# B&R Automation Studio project CleanChemi_SiteManagementSystem (part 7)

```iecst
		IF gSkid_LR[IdxSkids_LR].Alarms.ALARM_AB15.4 AND gServices.Alarms_LR[IdxSkids_LR].Internal.Alarms_State.ALARM_AB15.4 = FALSE THEN
			IF gSkid_LR[IdxSkids_LR].ErrorInfo.Text = '' THEN
				gSkid_LR[IdxSkids_LR].ErrorInfo.Text		:= 'ALARM_AB15.4';
				gSkid_LR[IdxSkids_LR].ErrorInfo.State		:= 'Warning';
				gSkid_LR[IdxSkids_LR].ErrorInfo.Severity	:= 1;
				gSkid_LR[IdxSkids_LR].Error := TRUE;
				gServices.Alarms_LR[IdxSkids_LR].Internal.Alarms_State.ALARM_AB15.4 := TRUE;
			END_IF
		END_IF;

		IF gSkid_LR[IdxSkids_LR].Alarms.ALARM_AB15.5 AND gServices.Alarms_LR[IdxSkids_LR].Internal.Alarms_State.ALARM_AB15.5 = FALSE THEN
			IF gSkid_LR[IdxSkids_LR].ErrorInfo.Text = '' THEN
				gSkid_LR[IdxSkids_LR].ErrorInfo.Text		:= 'ALARM_AB15.5';
				gSkid_LR[IdxSkids_LR].ErrorInfo.State		:= 'Warning';
				gSkid_LR[IdxSkids_LR].ErrorInfo.Severity	:= 1;
				gSkid_LR[IdxSkids_LR].Error := TRUE;
				gServices.Alarms_LR[IdxSkids_LR].Internal.Alarms_State.ALARM_AB15.5 := TRUE;
			END_IF
		END_IF;

		IF gSkid_LR[IdxSkids_LR].Alarms.ALARM_AB15.6 AND gServices.Alarms_LR[IdxSkids_LR].Internal.Alarms_State.ALARM_AB15.6 = FALSE THEN
			IF gSkid_LR[IdxSkids_LR].ErrorInfo.Text = '' THEN
				gSkid_LR[IdxSkids_LR].ErrorInfo.Text		:= 'ALARM_AB15.6';
				gSkid_LR[IdxSkids_LR].ErrorInfo.State		:= 'Warning';
				gSkid_LR[IdxSkids_LR].ErrorInfo.Severity	:= 1;
				gSkid_LR[IdxSkids_LR].Error := TRUE;
				gServices.Alarms_LR[IdxSkids_LR].Internal.Alarms_State.ALARM_AB15.6 := TRUE;
			END_IF
		END_IF;
		IF gSkid_LR[IdxSkids_LR].Alarms.ALARM_AB15.7 AND gServices.Alarms_LR[IdxSkids_LR].Internal.Alarms_State.ALARM_AB15.7 = FALSE THEN
			IF gSkid_LR[IdxSkids_LR].ErrorInfo.Text = '' THEN
				gSkid_LR[IdxSkids_LR].ErrorInfo.Text		:= 'ALARM_AB15.7';
				gSkid_LR[IdxSkids_LR].ErrorInfo.State		:= 'Warning';
				gSkid_LR[IdxSkids_LR].ErrorInfo.Severity	:= 1;
				gSkid_LR[IdxSkids_LR].Error := TRUE;
				gServices.Alarms_LR[IdxSkids_LR].Internal.Alarms_State.ALARM_AB15.7 := TRUE;
			END_IF
		END_IF;
		IF gSkid_LR[IdxSkids_LR].Alarms.ALARM_AB15.8 AND gServices.Alarms_LR[IdxSkids_LR].Internal.Alarms_State.ALARM_AB15.8 = FALSE THEN
			IF gSkid_LR[IdxSkids_LR].ErrorInfo.Text = '' THEN
				gSkid_LR[IdxSkids_LR].ErrorInfo.Text		:= 'ALARM_AB15.8';
				gSkid_LR[IdxSkids_LR].ErrorInfo.State		:= 'Warning';
				gSkid_LR[IdxSkids_LR].ErrorInfo.Severity	:= 1;
				gSkid_LR[IdxSkids_LR].Error := TRUE;
				gServices.Alarms_LR[IdxSkids_LR].Internal.Alarms_State.ALARM_AB15.8 := TRUE;
			END_IF
		END_IF;
		IF gSkid_LR[IdxSkids_LR].Alarms.ALARM_AB15.9 AND gServices.Alarms_LR[IdxSkids_LR].Internal.Alarms_State.ALARM_AB15.9 = FALSE THEN
			IF gSkid_LR[IdxSkids_LR].ErrorInfo.Text = '' THEN
				gSkid_LR[IdxSkids_LR].ErrorInfo.Text		:= 'ALARM_AB15.9';
				gSkid_LR[IdxSkids_LR].ErrorInfo.State		:= 'Warning';
				gSkid_LR[IdxSkids_LR].ErrorInfo.Severity	:= 1;
				gSkid_LR[IdxSkids_LR].Error := TRUE;
				gServices.Alarms_LR[IdxSkids_LR].Internal.Alarms_State.ALARM_AB15.9 := TRUE;
			END_IF
		END_IF;
		IF gSkid_LR[IdxSkids_LR].Alarms.ALARM_AB15.10 AND gServices.Alarms_LR[IdxSkids_LR].Internal.Alarms_State.ALARM_AB15.10 = FALSE THEN
			IF gSkid_LR[IdxSkids_LR].ErrorInfo.Text = '' THEN
				gSkid_LR[IdxSkids_LR].ErrorInfo.Text		:= 'ALARM_AB15.10';
				gSkid_LR[IdxSkids_LR].ErrorInfo.State		:= 'Warning';
				gSkid_LR[IdxSkids_LR].ErrorInfo.Severity	:= 1;
				gSkid_LR[IdxSkids_LR].Error := TRUE;
				gServices.Alarms_LR[IdxSkids_LR].Internal.Alarms_State.ALARM_AB15.10 := TRUE;
			END_IF
		END_IF;
		IF gSkid_LR[IdxSkids_LR].Alarms.ALARM_AB15.11 AND gServices.Alarms_LR[IdxSkids_LR].Internal.Alarms_State.ALARM_AB15.11 = FALSE THEN
			IF gSkid_LR[IdxSkids_LR].ErrorInfo.Text = '' THEN
				gSkid_LR[IdxSkids_LR].ErrorInfo.Text		:= 'ALARM_AB15.11';
				gSkid_LR[IdxSkids_LR].ErrorInfo.State		:= 'Warning';
				gSkid_LR[IdxSkids_LR].ErrorInfo.Severity	:= 1;
				gSkid_LR[IdxSkids_LR].Error := TRUE;
				gServices.Alarms_LR[IdxSkids_LR].Internal.Alarms_State.ALARM_AB15.11 := TRUE;
			END_IF
		END_IF;
		IF gSkid_LR[IdxSkids_LR].Alarms.ALARM_AB15.12 AND gServices.Alarms_LR[IdxSkids_LR].Internal.Alarms_State.ALARM_AB15.12 = FALSE THEN
			IF gSkid_LR[IdxSkids_LR].ErrorInfo.Text = '' THEN
				gSkid_LR[IdxSkids_LR].ErrorInfo.Text		:= 'ALARM_AB15.12';
				gSkid_LR[IdxSkids_LR].ErrorInfo.State		:= 'Warning';
				gSkid_LR[IdxSkids_LR].ErrorInfo.Severity	:= 1;
				gSkid_LR[IdxSkids_LR].Error := TRUE;
				gServices.Alarms_LR[IdxSkids_LR].Internal.Alarms_State.ALARM_AB15.12 := TRUE;
			END_IF
		END_IF;

		// AB16
		IF gSkid_LR[IdxSkids_LR].Alarms.ALARM_AB16.0 AND gServices.Alarms_LR[IdxSkids_LR].Internal.Alarms_State.ALARM_AB16.0 = FALSE THEN
			IF gSkid_LR[IdxSkids_LR].ErrorInfo.Text = '' THEN
				gSkid_LR[IdxSkids_LR].ErrorInfo.Text		:= 'ALARM_AB16.0';
				gSkid_LR[IdxSkids_LR].ErrorInfo.State		:= 'Warning';
				gSkid_LR[IdxSkids_LR].ErrorInfo.Severity	:= 2;
				gSkid_LR[IdxSkids_LR].Error := TRUE;
				gServices.Alarms_LR[IdxSkids_LR].Internal.Alarms_State.ALARM_AB16.0 := TRUE;
			END_IF
		END_IF;

		IF gSkid_LR[IdxSkids_LR].Alarms.ALARM_AB16.1 AND gServices.Alarms_LR[IdxSkids_LR].Internal.Alarms_State.ALARM_AB16.1 = FALSE THEN
			IF gSkid_LR[IdxSkids_LR].ErrorInfo.Text = '' THEN
				gSkid_LR[IdxSkids_LR].ErrorInfo.Text		:= 'ALARM_AB16.1';
				gSkid_LR[IdxSkids_LR].ErrorInfo.State		:= 'Warning';
				gSkid_LR[IdxSkids_LR].ErrorInfo.Severity	:= 1;
				gSkid_LR[IdxSkids_LR].Error := TRUE;
				gServices.Alarms_LR[IdxSkids_LR].Internal.Alarms_State.ALARM_AB16.1 := TRUE;
			END_IF
		END_IF;

		IF gSkid_LR[IdxSkids_LR].Alarms.ALARM_AB16.2 AND gServices.Alarms_LR[IdxSkids_LR].Internal.Alarms_State.ALARM_AB16.2 = FALSE THEN
			IF gSkid_LR[IdxSkids_LR].ErrorInfo.Text = '' THEN
				gSkid_LR[IdxSkids_LR].ErrorInfo.Text		:= 'ALARM_AB16.2';
				gSkid_LR[IdxSkids_LR].ErrorInfo.State		:= 'Warning';
				gSkid_LR[IdxSkids_LR].ErrorInfo.Severity	:= 2;
				gSkid_LR[IdxSkids_LR].Error := TRUE;
				gServices.Alarms_LR[IdxSkids_LR].Internal.Alarms_State.ALARM_AB16.2 := TRUE;
			END_IF
		END_IF;

		IF gSkid_LR[IdxSkids_LR].Alarms.ALARM_AB16.3 AND gServices.Alarms_LR[IdxSkids_LR].Internal.Alarms_State.ALARM_AB16.3 = FALSE THEN
			IF gSkid_LR[IdxSkids_LR].ErrorInfo.Text = '' THEN
				gSkid_LR[IdxSkids_LR].ErrorInfo.Text		:= 'ALARM_AB16.3';
				gSkid_LR[IdxSkids_LR].ErrorInfo.State		:= 'Warning';
				gSkid_LR[IdxSkids_LR].ErrorInfo.Severity	:= 1;
				gSkid_LR[IdxSkids_LR].Error := TRUE;
				gServices.Alarms_LR[IdxSkids_LR].Internal.Alarms_State.ALARM_AB16.3 := TRUE;
			END_IF
		END_IF;

		IF gSkid_LR[IdxSkids_LR].Alarms.ALARM_AB16.4 AND gServices.Alarms_LR[IdxSkids_LR].Internal.Alarms_State.ALARM_AB16.4 = FALSE THEN
			IF gSkid_LR[IdxSkids_LR].ErrorInfo.Text = '' THEN
				gSkid_LR[IdxSkids_LR].ErrorInfo.Text		:= 'ALARM_AB16.4';
				gSkid_LR[IdxSkids_LR].ErrorInfo.State		:= 'Warning';
				gSkid_LR[IdxSkids_LR].ErrorInfo.Severity	:= 2;
				gSkid_LR[IdxSkids_LR].Error := TRUE;
				gServices.Alarms_LR[IdxSkids_LR].Internal.Alarms_State.ALARM_AB16.4 := TRUE;
			END_IF
		END_IF;

		IF gSkid_LR[IdxSkids_LR].Alarms.ALARM_AB16.5 AND gServices.Alarms_LR[IdxSkids_LR].Internal.Alarms_State.ALARM_AB16.5 = FALSE THEN
			IF gSkid_LR[IdxSkids_LR].ErrorInfo.Text = '' THEN
				gSkid_LR[IdxSkids_LR].ErrorInfo.Text		:= 'ALARM_AB16.5';
				gSkid_LR[IdxSkids_LR].ErrorInfo.State		:= 'Warning';
				gSkid_LR[IdxSkids_LR].ErrorInfo.Severity	:= 1;
				gSkid_LR[IdxSkids_LR].Error := TRUE;
				gServices.Alarms_LR[IdxSkids_LR].Internal.Alarms_State.ALARM_AB16.5 := TRUE;
			END_IF
		END_IF;

		IF gSkid_LR[IdxSkids_LR].Alarms.ALARM_AB16.6 AND gServices.Alarms_LR[IdxSkids_LR].Internal.Alarms_State.ALARM_AB16.6 = FALSE THEN
			IF gSkid_LR[IdxSkids_LR].ErrorInfo.Text = '' THEN
				gSkid_LR[IdxSkids_LR].ErrorInfo.Text		:= 'ALARM_AB16.6';
				gSkid_LR[IdxSkids_LR].ErrorInfo.State		:= 'Warning';
				gSkid_LR[IdxSkids_LR].ErrorInfo.Severity	:= 2;
				gSkid_LR[IdxSkids_LR].Error := TRUE;
				gServices.Alarms_LR[IdxSkids_LR].Internal.Alarms_State.ALARM_AB16.6 := TRUE;
			END_IF
		END_IF;
		IF gSkid_LR[IdxSkids_LR].Alarms.ALARM_AB16.7 AND gServices.Alarms_LR[IdxSkids_LR].Internal.Alarms_State.ALARM_AB16.7 = FALSE THEN
			IF gSkid_LR[IdxSkids_LR].ErrorInfo.Text = '' THEN
				gSkid_LR[IdxSkids_LR].ErrorInfo.Text		:= 'ALARM_AB16.7';
				gSkid_LR[IdxSkids_LR].ErrorInfo.State		:= 'Warning';
				gSkid_LR[IdxSkids_LR].ErrorInfo.Severity	:= 1;
				gSkid_LR[IdxSkids_LR].Error := TRUE;
				gServices.Alarms_LR[IdxSkids_LR].Internal.Alarms_State.ALARM_AB16.7 := TRUE;
			END_IF
		END_IF;
		IF gSkid_LR[IdxSkids_LR].Alarms.ALARM_AB16.8 AND gServices.Alarms_LR[IdxSkids_LR].Internal.Alarms_State.ALARM_AB16.8 = FALSE THEN
			IF gSkid_LR[IdxSkids_LR].ErrorInfo.Text = '' THEN
				gSkid_LR[IdxSkids_LR].ErrorInfo.Text		:= 'ALARM_AB16.8';
				gSkid_LR[IdxSkids_LR].ErrorInfo.State		:= 'Warning';
				gSkid_LR[IdxSkids_LR].ErrorInfo.Severity	:= 2;
				gSkid_LR[IdxSkids_LR].Error := TRUE;
				gServices.Alarms_LR[IdxSkids_LR].Internal.Alarms_State.ALARM_AB16.8 := TRUE;
			END_IF
		END_IF;
		IF gSkid_LR[IdxSkids_LR].Alarms.ALARM_AB16.9 AND gServices.Alarms_LR[IdxSkids_LR].Internal.Alarms_State.ALARM_AB16.9 = FALSE THEN
			IF gSkid_LR[IdxSkids_LR].ErrorInfo.Text = '' THEN
				gSkid_LR[IdxSkids_LR].ErrorInfo.Text		:= 'ALARM_AB16.9';
				gSkid_LR[IdxSkids_LR].ErrorInfo.State		:= 'Warning';
				gSkid_LR[IdxSkids_LR].ErrorInfo.Severity	:= 1;
				gSkid_LR[IdxSkids_LR].Error := TRUE;
				gServices.Alarms_LR[IdxSkids_LR].Internal.Alarms_State.ALARM_AB16.9 := TRUE;
			END_IF
		END_IF;
		IF gSkid_LR[IdxSkids_LR].Alarms.ALARM_AB16.10 AND gServices.Alarms_LR[IdxSkids_LR].Internal.Alarms_State.ALARM_AB16.10 = FALSE THEN
			IF gSkid_LR[IdxSkids_LR].ErrorInfo.Text = '' THEN
				gSkid_LR[IdxSkids_LR].ErrorInfo.Text		:= 'ALARM_AB16.10';
				gSkid_LR[IdxSkids_LR].ErrorInfo.State		:= 'Warning';
				gSkid_LR[IdxSkids_LR].ErrorInfo.Severity	:= 2;
				gSkid_LR[IdxSkids_LR].Error := TRUE;
				gServices.Alarms_LR[IdxSkids_LR].Internal.Alarms_State.ALARM_AB16.10 := TRUE;
			END_IF
		END_IF;
		IF gSkid_LR[IdxSkids_LR].Alarms.ALARM_AB16.11 AND gServices.Alarms_LR[IdxSkids_LR].Internal.Alarms_State.ALARM_AB16.11 = FALSE THEN
			IF gSkid_LR[IdxSkids_LR].ErrorInfo.Text = '' THEN
				gSkid_LR[IdxSkids_LR].ErrorInfo.Text		:= 'ALARM_AB16.11';
				gSkid_LR[IdxSkids_LR].ErrorInfo.State		:= 'Warning';
				gSkid_LR[IdxSkids_LR].ErrorInfo.Severity	:= 1;
				gSkid_LR[IdxSkids_LR].Error := TRUE;
				gServices.Alarms_LR[IdxSkids_LR].Internal.Alarms_State.ALARM_AB16.11 := TRUE;
			END_IF
		END_IF;
		IF gSkid_LR[IdxSkids_LR].Alarms.ALARM_AB16.12 AND gServices.Alarms_LR[IdxSkids_LR].Internal.Alarms_State.ALARM_AB16.12 = FALSE THEN
			IF gSkid_LR[IdxSkids_LR].ErrorInfo.Text = '' THEN
				gSkid_LR[IdxSkids_LR].ErrorInfo.Text		:= 'ALARM_AB16.12';
				gSkid_LR[IdxSkids_LR].ErrorInfo.State		:= 'Warning';
				gSkid_LR[IdxSkids_LR].ErrorInfo.Severity	:= 2;
				gSkid_LR[IdxSkids_LR].Error := TRUE;
				gServices.Alarms_LR[IdxSkids_LR].Internal.Alarms_State.ALARM_AB16.12 := TRUE;
			END_IF
		END_IF;
		IF gSkid_LR[IdxSkids_LR].Alarms.ALARM_AB16.13 AND gServices.Alarms_LR[IdxSkids_LR].Internal.Alarms_State.ALARM_AB16.13 = FALSE THEN
			IF gSkid_LR[IdxSkids_LR].ErrorInfo.Text = '' THEN
				gSkid_LR[IdxSkids_LR].ErrorInfo.Text		:= 'ALARM_AB16.13';
				gSkid_LR[IdxSkids_LR].ErrorInfo.State		:= 'Warning';
				gSkid_LR[IdxSkids_LR].ErrorInfo.Severity	:= 1;
				gSkid_LR[IdxSkids_LR].Error := TRUE;
				gServices.Alarms_LR[IdxSkids_LR].Internal.Alarms_State.ALARM_AB16.13 := TRUE;
			END_IF
		END_IF;
		IF gSkid_LR[IdxSkids_LR].Alarms.ALARM_AB16.14 AND gServices.Alarms_LR[IdxSkids_LR].Internal.Alarms_State.ALARM_AB16.14 = FALSE THEN
			IF gSkid_LR[IdxSkids_LR].ErrorInfo.Text = '' THEN
				gSkid_LR[IdxSkids_LR].ErrorInfo.Text		:= 'ALARM_AB16.14';
				gSkid_LR[IdxSkids_LR].ErrorInfo.State		:= 'Warning';
				gSkid_LR[IdxSkids_LR].ErrorInfo.Severity	:= 2;
				gSkid_LR[IdxSkids_LR].Error := TRUE;
				gServices.Alarms_LR[IdxSkids_LR].Internal.Alarms_State.ALARM_AB16.14 := TRUE;
			END_IF
		END_IF;
		IF gSkid_LR[IdxSkids_LR].Alarms.ALARM_AB16.15 AND gServices.Alarms_LR[IdxSkids_LR].Internal.Alarms_State.ALARM_AB16.15 = FALSE THEN
			IF gSkid_LR[IdxSkids_LR].ErrorInfo.Text = '' THEN
				gSkid_LR[IdxSkids_LR].ErrorInfo.Text		:= 'ALARM_AB16.15';
				gSkid_LR[IdxSkids_LR].ErrorInfo.State		:= 'Warning';
				gSkid_LR[IdxSkids_LR].ErrorInfo.Severity	:= 1;
				gSkid_LR[IdxSkids_LR].Error := TRUE;
				gServices.Alarms_LR[IdxSkids_LR].Internal.Alarms_State.ALARM_AB16.15 := TRUE;
			END_IF
		END_IF;

		// AB17
		IF gSkid_LR[IdxSkids_LR].Alarms.ALARM_AB17.0 AND gServices.Alarms_LR[IdxSkids_LR].Internal.Alarms_State.ALARM_AB17.0 = FALSE THEN
			IF gSkid_LR[IdxSkids_LR].ErrorInfo.Text = '' THEN
				gSkid_LR[IdxSkids_LR].ErrorInfo.Text		:= 'ALARM_AB17.0';
				gSkid_LR[IdxSkids_LR].ErrorInfo.State		:= 'Warning';
				gSkid_LR[IdxSkids_LR].ErrorInfo.Severity	:= 2;
				gSkid_LR[IdxSkids_LR].Error := TRUE;
				gServices.Alarms_LR[IdxSkids_LR].Internal.Alarms_State.ALARM_AB17.0 := TRUE;
			END_IF
		END_IF;

		IF gSkid_LR[IdxSkids_LR].Alarms.ALARM_AB17.1 AND gServices.Alarms_LR[IdxSkids_LR].Internal.Alarms_State.ALARM_AB17.1 = FALSE THEN
			IF gSkid_LR[IdxSkids_LR].ErrorInfo.Text = '' THEN
				gSkid_LR[IdxSkids_LR].ErrorInfo.Text		:= 'ALARM_AB17.1';
				gSkid_LR[IdxSkids_LR].ErrorInfo.State		:= 'Warning';
				gSkid_LR[IdxSkids_LR].ErrorInfo.Severity	:= 1;
				gSkid_LR[IdxSkids_LR].Error := TRUE;
				gServices.Alarms_LR[IdxSkids_LR].Internal.Alarms_State.ALARM_AB17.1 := TRUE;
			END_IF
		END_IF;

		IF gSkid_LR[IdxSkids_LR].Alarms.ALARM_AB17.2 AND gServices.Alarms_LR[IdxSkids_LR].Internal.Alarms_State.ALARM_AB17.2 = FALSE THEN
			IF gSkid_LR[IdxSkids_LR].ErrorInfo.Text = '' THEN
				gSkid_LR[IdxSkids_LR].ErrorInfo.Text		:= 'ALARM_AB17.2';
				gSkid_LR[IdxSkids_LR].ErrorInfo.State		:= 'Warning';
				gSkid_LR[IdxSkids_LR].ErrorInfo.Severity	:= 1;
				gSkid_LR[IdxSkids_LR].Error := TRUE;
				gServices.Alarms_LR[IdxSkids_LR].Internal.Alarms_State.ALARM_AB17.2 := TRUE;
			END_IF
		END_IF;

		IF gSkid_LR[IdxSkids_LR].Alarms.ALARM_AB17.3 AND gServices.Alarms_LR[IdxSkids_LR].Internal.Alarms_State.ALARM_AB17.3 = FALSE THEN
			IF gSkid_LR[IdxSkids_LR].ErrorInfo.Text = '' THEN
				gSkid_LR[IdxSkids_LR].ErrorInfo.Text		:= 'ALARM_AB17.3';
				gSkid_LR[IdxSkids_LR].ErrorInfo.State		:= 'Warning';
				gSkid_LR[IdxSkids_LR].ErrorInfo.Severity	:= 1;
				gSkid_LR[IdxSkids_LR].Error := TRUE;
				gServices.Alarms_LR[IdxSkids_LR].Internal.Alarms_State.ALARM_AB17.3 := TRUE;
			END_IF
		END_IF;

		IF gSkid_LR[IdxSkids_LR].Alarms.ALARM_AB17.4 AND gServices.Alarms_LR[IdxSkids_LR].Internal.Alarms_State.ALARM_AB17.4 = FALSE THEN
			IF gSkid_LR[IdxSkids_LR].ErrorInfo.Text = '' THEN
				gSkid_LR[IdxSkids_LR].ErrorInfo.Text		:= 'ALARM_AB17.4';
				gSkid_LR[IdxSkids_LR].ErrorInfo.State		:= 'Warning';
				gSkid_LR[IdxSkids_LR].ErrorInfo.Severity	:= 1;
				gSkid_LR[IdxSkids_LR].Error := TRUE;
				gServices.Alarms_LR[IdxSkids_LR].Internal.Alarms_State.ALARM_AB17.4 := TRUE;
			END_IF
		END_IF;

		IF gSkid_LR[IdxSkids_LR].Alarms.ALARM_AB17.5 AND gServices.Alarms_LR[IdxSkids_LR].Internal.Alarms_State.ALARM_AB17.5 = FALSE THEN
			IF gSkid_LR[IdxSkids_LR].ErrorInfo.Text = '' THEN
				gSkid_LR[IdxSkids_LR].ErrorInfo.Text		:= 'ALARM_AB17.5';
				gSkid_LR[IdxSkids_LR].ErrorInfo.State		:= 'Warning';
				gSkid_LR[IdxSkids_LR].ErrorInfo.Severity	:= 1;
				gSkid_LR[IdxSkids_LR].Error := TRUE;
				gServices.Alarms_LR[IdxSkids_LR].Internal.Alarms_State.ALARM_AB17.5 := TRUE;
			END_IF
		END_IF;

		IF gSkid_LR[IdxSkids_LR].Alarms.ALARM_AB17.6 AND gServices.Alarms_LR[IdxSkids_LR].Internal.Alarms_State.ALARM_AB17.6 = FALSE THEN
			IF gSkid_LR[IdxSkids_LR].ErrorInfo.Text = '' THEN
				gSkid_LR[IdxSkids_LR].ErrorInfo.Text		:= 'ALARM_AB17.6';
				gSkid_LR[IdxSkids_LR].ErrorInfo.State		:= 'Warning';
				gSkid_LR[IdxSkids_LR].ErrorInfo.Severity	:= 1;
				gSkid_LR[IdxSkids_LR].Error := TRUE;
				gServices.Alarms_LR[IdxSkids_LR].Internal.Alarms_State.ALARM_AB17.6 := TRUE;
			END_IF
		END_IF;
		IF gSkid_LR[IdxSkids_LR].Alarms.ALARM_AB17.7 AND gServices.Alarms_LR[IdxSkids_LR].Internal.Alarms_State.ALARM_AB17.7 = FALSE THEN
			IF gSkid_LR[IdxSkids_LR].ErrorInfo.Text = '' THEN
				gSkid_LR[IdxSkids_LR].ErrorInfo.Text		:= 'ALARM_AB17.7';
				gSkid_LR[IdxSkids_LR].ErrorInfo.State		:= 'Warning';
				gSkid_LR[IdxSkids_LR].ErrorInfo.Severity	:= 1;
				gSkid_LR[IdxSkids_LR].Error := TRUE;
				gServices.Alarms_LR[IdxSkids_LR].Internal.Alarms_State.ALARM_AB17.7 := TRUE;
			END_IF
		END_IF;
		IF gSkid_LR[IdxSkids_LR].Alarms.ALARM_AB17.8 AND gServices.Alarms_LR[IdxSkids_LR].Internal.Alarms_State.ALARM_AB17.8 = FALSE THEN
			IF gSkid_LR[IdxSkids_LR].ErrorInfo.Text = '' THEN
				gSkid_LR[IdxSkids_LR].ErrorInfo.Text		:= 'ALARM_AB17.8';
				gSkid_LR[IdxSkids_LR].ErrorInfo.State		:= 'Warning';
				gSkid_LR[IdxSkids_LR].ErrorInfo.Severity	:= 1;
				gSkid_LR[IdxSkids_LR].Error := TRUE;
				gServices.Alarms_LR[IdxSkids_LR].Internal.Alarms_State.ALARM_AB17.8 := TRUE;
			END_IF
		END_IF;
		IF gSkid_LR[IdxSkids_LR].Alarms.ALARM_AB17.9 AND gServices.Alarms_LR[IdxSkids_LR].Internal.Alarms_State.ALARM_AB17.9 = FALSE THEN
			IF gSkid_LR[IdxSkids_LR].ErrorInfo.Text = '' THEN
				gSkid_LR[IdxSkids_LR].ErrorInfo.Text		:= 'ALARM_AB17.9';
				gSkid_LR[IdxSkids_LR].ErrorInfo.State		:= 'Warning';
				gSkid_LR[IdxSkids_LR].ErrorInfo.Severity	:= 1;
				gSkid_LR[IdxSkids_LR].Error := TRUE;
				gServices.Alarms_LR[IdxSkids_LR].Internal.Alarms_State.ALARM_AB17.9 := TRUE;
			END_IF
		END_IF;
		IF gSkid_LR[IdxSkids_LR].Alarms.ALARM_AB17.10 AND gServices.Alarms_LR[IdxSkids_LR].Internal.Alarms_State.ALARM_AB17.10 = FALSE THEN
			IF gSkid_LR[IdxSkids_LR].ErrorInfo.Text = '' THEN
				gSkid_LR[IdxSkids_LR].ErrorInfo.Text		:= 'ALARM_AB17.10';
				gSkid_LR[IdxSkids_LR].ErrorInfo.State		:= 'Warning';
				gSkid_LR[IdxSkids_LR].ErrorInfo.Severity	:= 1;
				gSkid_LR[IdxSkids_LR].Error := TRUE;
				gServices.Alarms_LR[IdxSkids_LR].Internal.Alarms_State.ALARM_AB17.10 := TRUE;
			END_IF
		END_IF;
		IF gSkid_LR[IdxSkids_LR].Alarms.ALARM_AB17.11 AND gServices.Alarms_LR[IdxSkids_LR].Internal.Alarms_State.ALARM_AB17.11 = FALSE THEN
			IF gSkid_LR[IdxSkids_LR].ErrorInfo.Text = '' THEN
				gSkid_LR[IdxSkids_LR].ErrorInfo.Text		:= 'ALARM_AB17.11';
				gSkid_LR[IdxSkids_LR].ErrorInfo.State		:= 'Warning';
				gSkid_LR[IdxSkids_LR].ErrorInfo.Severity	:= 1;
				gSkid_LR[IdxSkids_LR].Error := TRUE;
				gServices.Alarms_LR[IdxSkids_LR].Internal.Alarms_State.ALARM_AB17.11 := TRUE;
			END_IF
		END_IF;
		IF gSkid_LR[IdxSkids_LR].Alarms.ALARM_AB17.12 AND gServices.Alarms_LR[IdxSkids_LR].Internal.Alarms_State.ALARM_AB17.12 = FALSE THEN
			IF gSkid_LR[IdxSkids_LR].ErrorInfo.Text = '' THEN
				gSkid_LR[IdxSkids_LR].ErrorInfo.Text		:= 'ALARM_AB17.12';
				gSkid_LR[IdxSkids_LR].ErrorInfo.State		:= 'Warning';
				gSkid_LR[IdxSkids_LR].ErrorInfo.Severity	:= 1;
				gSkid_LR[IdxSkids_LR].Error := TRUE;
				gServices.Alarms_LR[IdxSkids_LR].Internal.Alarms_State.ALARM_AB17.12 := TRUE;
			END_IF
		END_IF;

		// AB18
		IF gSkid_LR[IdxSkids_LR].Alarms.ALARM_AB18.0 AND gServices.Alarms_LR[IdxSkids_LR].Internal.Alarms_State.ALARM_AB18.0 = FALSE THEN
			IF gSkid_LR[IdxSkids_LR].ErrorInfo.Text = '' THEN
				gSkid_LR[IdxSkids_LR].ErrorInfo.Text		:= 'ALARM_AB18.0';
				gSkid_LR[IdxSkids_LR].ErrorInfo.State		:= 'Warning';
				gSkid_LR[IdxSkids_LR].ErrorInfo.Severity	:= 2;
				gSkid_LR[IdxSkids_LR].Error := TRUE;
				gServices.Alarms_LR[IdxSkids_LR].Internal.Alarms_State.ALARM_AB18.0 := TRUE;
			END_IF
		END_IF;

		IF gSkid_LR[IdxSkids_LR].Alarms.ALARM_AB18.1 AND gServices.Alarms_LR[IdxSkids_LR].Internal.Alarms_State.ALARM_AB18.1 = FALSE THEN
			IF gSkid_LR[IdxSkids_LR].ErrorInfo.Text = '' THEN
				gSkid_LR[IdxSkids_LR].ErrorInfo.Text		:= 'ALARM_AB18.1';
				gSkid_LR[IdxSkids_LR].ErrorInfo.State		:= 'Warning';
				gSkid_LR[IdxSkids_LR].ErrorInfo.Severity	:= 1;
				gSkid_LR[IdxSkids_LR].Error := TRUE;
				gServices.Alarms_LR[IdxSkids_LR].Internal.Alarms_State.ALARM_AB18.1 := TRUE;
			END_IF
		END_IF;

		IF gSkid_LR[IdxSkids_LR].Alarms.ALARM_AB18.2 AND gServices.Alarms_LR[IdxSkids_LR].Internal.Alarms_State.ALARM_AB18.2 = FALSE THEN
			IF gSkid_LR[IdxSkids_LR].ErrorInfo.Text = '' THEN
				gSkid_LR[IdxSkids_LR].ErrorInfo.Text		:= 'ALARM_AB18.2';
				gSkid_LR[IdxSkids_LR].ErrorInfo.State		:= 'Warning';
				gSkid_LR[IdxSkids_LR].ErrorInfo.Severity	:= 2;
				gSkid_LR[IdxSkids_LR].Error := TRUE;
				gServices.Alarms_LR[IdxSkids_LR].Internal.Alarms_State.ALARM_AB18.2 := TRUE;
			END_IF
		END_IF;

		IF gSkid_LR[IdxSkids_LR].Alarms.ALARM_AB18.3 AND gServices.Alarms_LR[IdxSkids_LR].Internal.Alarms_State.ALARM_AB18.3 = FALSE THEN
			IF gSkid_LR[IdxSkids_LR].ErrorInfo.Text = '' THEN
				gSkid_LR[IdxSkids_LR].ErrorInfo.Text		:= 'ALARM_AB18.3';
				gSkid_LR[IdxSkids_LR].ErrorInfo.State		:= 'Warning';
				gSkid_LR[IdxSkids_LR].ErrorInfo.Severity	:= 1;
				gSkid_LR[IdxSkids_LR].Error := TRUE;
				gServices.Alarms_LR[IdxSkids_LR].Internal.Alarms_State.ALARM_AB18.3 := TRUE;
			END_IF
		END_IF;

		IF gSkid_LR[IdxSkids_LR].Alarms.ALARM_AB18.4 AND gServices.Alarms_LR[IdxSkids_LR].Internal.Alarms_State.ALARM_AB18.4 = FALSE THEN
			IF gSkid_LR[IdxSkids_LR].ErrorInfo.Text = '' THEN
				gSkid_LR[IdxSkids_LR].ErrorInfo.Text		:= 'ALARM_AB18.4';
				gSkid_LR[IdxSkids_LR].ErrorInfo.State		:= 'Warning';
				gSkid_LR[IdxSkids_LR].ErrorInfo.Severity	:= 2;
				gSkid_LR[IdxSkids_LR].Error := TRUE;
				gServices.Alarms_LR[IdxSkids_LR].Internal.Alarms_State.ALARM_AB18.4 := TRUE;
			END_IF
		END_IF;

		IF gSkid_LR[IdxSkids_LR].Alarms.ALARM_AB18.5 AND gServices.Alarms_LR[IdxSkids_LR].Internal.Alarms_State.ALARM_AB18.5 = FALSE THEN
			IF gSkid_LR[IdxSkids_LR].ErrorInfo.Text = '' THEN
				gSkid_LR[IdxSkids_LR].ErrorInfo.Text		:= 'ALARM_AB18.5';
				gSkid_LR[IdxSkids_LR].ErrorInfo.State		:= 'Warning';
				gSkid_LR[IdxSkids_LR].ErrorInfo.Severity	:= 1;
				gSkid_LR[IdxSkids_LR].Error := TRUE;
				gServices.Alarms_LR[IdxSkids_LR].Internal.Alarms_State.ALARM_AB18.5 := TRUE;
			END_IF
		END_IF;

		IF gSkid_LR[IdxSkids_LR].Alarms.ALARM_AB18.6 AND gServices.Alarms_LR[IdxSkids_LR].Internal.Alarms_State.ALARM_AB18.6 = FALSE THEN
			IF gSkid_LR[IdxSkids_LR].ErrorInfo.Text = '' THEN
				gSkid_LR[IdxSkids_LR].ErrorInfo.Text		:= 'ALARM_AB18.6';
				gSkid_LR[IdxSkids_LR].ErrorInfo.State		:= 'Warning';
				gSkid_LR[IdxSkids_LR].ErrorInfo.Severity	:= 2;
				gSkid_LR[IdxSkids_LR].Error := TRUE;
				gServices.Alarms_LR[IdxSkids_LR].Internal.Alarms_State.ALARM_AB18.6 := TRUE;
			END_IF
		END_IF;
		IF gSkid_LR[IdxSkids_LR].Alarms.ALARM_AB18.7 AND gServices.Alarms_LR[IdxSkids_LR].Internal.Alarms_State.ALARM_AB18.7 = FALSE THEN
			IF gSkid_LR[IdxSkids_LR].ErrorInfo.Text = '' THEN
				gSkid_LR[IdxSkids_LR].ErrorInfo.Text		:= 'ALARM_AB18.7';
				gSkid_LR[IdxSkids_LR].ErrorInfo.State		:= 'Warning';
				gSkid_LR[IdxSkids_LR].ErrorInfo.Severity	:= 1;
				gSkid_LR[IdxSkids_LR].Error := TRUE;
				gServices.Alarms_LR[IdxSkids_LR].Internal.Alarms_State.ALARM_AB18.7 := TRUE;
			END_IF
		END_IF;
		IF gSkid_LR[IdxSkids_LR].Alarms.ALARM_AB18.8 AND gServices.Alarms_LR[IdxSkids_LR].Internal.Alarms_State.ALARM_AB18.8 = FALSE THEN
			IF gSkid_LR[IdxSkids_LR].ErrorInfo.Text = '' THEN
				gSkid_LR[IdxSkids_LR].ErrorInfo.Text		:= 'ALARM_AB18.8';
				gSkid_LR[IdxSkids_LR].ErrorInfo.State		:= 'Warning';
				gSkid_LR[IdxSkids_LR].ErrorInfo.Severity	:= 2;
				gSkid_LR[IdxSkids_LR].Error := TRUE;
				gServices.Alarms_LR[IdxSkids_LR].Internal.Alarms_State.ALARM_AB18.8 := TRUE;
			END_IF
		END_IF;
		IF gSkid_LR[IdxSkids_LR].Alarms.ALARM_AB18.9 AND gServices.Alarms_LR[IdxSkids_LR].Internal.Alarms_State.ALARM_AB18.9 = FALSE THEN
			IF gSkid_LR[IdxSkids_LR].ErrorInfo.Text = '' THEN
				gSkid_LR[IdxSkids_LR].ErrorInfo.Text		:= 'ALARM_AB18.9';
				gSkid_LR[IdxSkids_LR].ErrorInfo.State		:= 'Warning';
				gSkid_LR[IdxSkids_LR].ErrorInfo.Severity	:= 1;
				gSkid_LR[IdxSkids_LR].Error := TRUE;
				gServices.Alarms_LR[IdxSkids_LR].Internal.Alarms_State.ALARM_AB18.9 := TRUE;
			END_IF
		END_IF;
		IF gSkid_LR[IdxSkids_LR].Alarms.ALARM_AB18.10 AND gServices.Alarms_LR[IdxSkids_LR].Internal.Alarms_State.ALARM_AB18.10 = FALSE THEN
			IF gSkid_LR[IdxSkids_LR].ErrorInfo.Text = '' THEN
				gSkid_LR[IdxSkids_LR].ErrorInfo.Text		:= 'ALARM_AB18.10';
				gSkid_LR[IdxSkids_LR].ErrorInfo.State		:= 'Warning';
				gSkid_LR[IdxSkids_LR].ErrorInfo.Severity	:= 2;
				gSkid_LR[IdxSkids_LR].Error := TRUE;
				gServices.Alarms_LR[IdxSkids_LR].Internal.Alarms_State.ALARM_AB18.10 := TRUE;
			END_IF
		END_IF;
		IF gSkid_LR[IdxSkids_LR].Alarms.ALARM_AB18.11 AND gServices.Alarms_LR[IdxSkids_LR].Internal.Alarms_State.ALARM_AB18.11 = FALSE THEN
			IF gSkid_LR[IdxSkids_LR].ErrorInfo.Text = '' THEN
				gSkid_LR[IdxSkids_LR].ErrorInfo.Text		:= 'ALARM_AB18.11';
				gSkid_LR[IdxSkids_LR].ErrorInfo.State		:= 'Warning';
				gSkid_LR[IdxSkids_LR].ErrorInfo.Severity	:= 1;
				gSkid_LR[IdxSkids_LR].Error := TRUE;
				gServices.Alarms_LR[IdxSkids_LR].Internal.Alarms_State.ALARM_AB18.11 := TRUE;
			END_IF
		END_IF;
		IF gSkid_LR[IdxSkids_LR].Alarms.ALARM_AB18.12 AND gServices.Alarms_LR[IdxSkids_LR].Internal.Alarms_State.ALARM_AB18.12 = FALSE THEN
			IF gSkid_LR[IdxSkids_LR].ErrorInfo.Text = '' THEN
				gSkid_LR[IdxSkids_LR].ErrorInfo.Text		:= 'ALARM_AB18.12';
				gSkid_LR[IdxSkids_LR].ErrorInfo.State		:= 'Warning';
				gSkid_LR[IdxSkids_LR].ErrorInfo.Severity	:= 2;
				gSkid_LR[IdxSkids_LR].Error := TRUE;
				gServices.Alarms_LR[IdxSkids_LR].Internal.Alarms_State.ALARM_AB18.12 := TRUE;
			END_IF
		END_IF;
		IF gSkid_LR[IdxSkids_LR].Alarms.ALARM_AB18.13 AND gServices.Alarms_LR[IdxSkids_LR].Internal.Alarms_State.ALARM_AB18.13 = FALSE THEN
			IF gSkid_LR[IdxSkids_LR].ErrorInfo.Text = '' THEN
				gSkid_LR[IdxSkids_LR].ErrorInfo.Text		:= 'ALARM_AB18.13';
				gSkid_LR[IdxSkids_LR].ErrorInfo.State		:= 'Warning';
				gSkid_LR[IdxSkids_LR].ErrorInfo.Severity	:= 1;
				gSkid_LR[IdxSkids_LR].Error := TRUE;
				gServices.Alarms_LR[IdxSkids_LR].Internal.Alarms_State.ALARM_AB18.13 := TRUE;
			END_IF
		END_IF;
		IF gSkid_LR[IdxSkids_LR].Alarms.ALARM_AB18.14 AND gServices.Alarms_LR[IdxSkids_LR].Internal.Alarms_State.ALARM_AB18.14 = FALSE THEN
			IF gSkid_LR[IdxSkids_LR].ErrorInfo.Text = '' THEN
				gSkid_LR[IdxSkids_LR].ErrorInfo.Text		:= 'ALARM_AB18.14';
				gSkid_LR[IdxSkids_LR].ErrorInfo.State		:= 'Warning';
				gSkid_LR[IdxSkids_LR].ErrorInfo.Severity	:= 2;
				gSkid_LR[IdxSkids_LR].Error := TRUE;
				gServices.Alarms_LR[IdxSkids_LR].Internal.Alarms_State.ALARM_AB18.14 := TRUE;
			END_IF
		END_IF;
		IF gSkid_LR[IdxSkids_LR].Alarms.ALARM_AB18.15 AND gServices.Alarms_LR[IdxSkids_LR].Internal.Alarms_State.ALARM_AB18.15 = FALSE THEN
			IF gSkid_LR[IdxSkids_LR].ErrorInfo.Text = '' THEN
				gSkid_LR[IdxSkids_LR].ErrorInfo.Text		:= 'ALARM_AB18.15';
				gSkid_LR[IdxSkids_LR].ErrorInfo.State		:= 'Warning';
				gSkid_LR[IdxSkids_LR].ErrorInfo.Severity	:= 1;
				gSkid_LR[IdxSkids_LR].Error := TRUE;
				gServices.Alarms_LR[IdxSkids_LR].Internal.Alarms_State.ALARM_AB18.15 := TRUE;
			END_IF
		END_IF;

		// AB19
		IF gSkid_LR[IdxSkids_LR].Alarms.ALARM_AB19.0 AND gServices.Alarms_LR[IdxSkids_LR].Internal.Alarms_State.ALARM_AB19.0 = FALSE THEN
			IF gSkid_LR[IdxSkids_LR].ErrorInfo.Text = '' THEN
				gSkid_LR[IdxSkids_LR].ErrorInfo.Text		:= 'ALARM_AB19.0';
				gSkid_LR[IdxSkids_LR].ErrorInfo.State		:= 'Warning';
				gSkid_LR[IdxSkids_LR].ErrorInfo.Severity	:= 2;
				gSkid_LR[IdxSkids_LR].Error := TRUE;
				gServices.Alarms_LR[IdxSkids_LR].Internal.Alarms_State.ALARM_AB19.0 := TRUE;
			END_IF
		END_IF;

		IF gSkid_LR[IdxSkids_LR].Alarms.ALARM_AB19.1 AND gServices.Alarms_LR[IdxSkids_LR].Internal.Alarms_State.ALARM_AB19.1 = FALSE THEN
			IF gSkid_LR[IdxSkids_LR].ErrorInfo.Text = '' THEN
				gSkid_LR[IdxSkids_LR].ErrorInfo.Text		:= 'ALARM_AB19.1';
				gSkid_LR[IdxSkids_LR].ErrorInfo.State		:= 'Warning';
				gSkid_LR[IdxSkids_LR].ErrorInfo.Severity	:= 1;
				gSkid_LR[IdxSkids_LR].Error := TRUE;
				gServices.Alarms_LR[IdxSkids_LR].Internal.Alarms_State.ALARM_AB19.1 := TRUE;
			END_IF
		END_IF;

		IF gSkid_LR[IdxSkids_LR].Alarms.ALARM_AB19.2 AND gServices.Alarms_LR[IdxSkids_LR].Internal.Alarms_State.ALARM_AB19.2 = FALSE THEN
			IF gSkid_LR[IdxSkids_LR].ErrorInfo.Text = '' THEN
				gSkid_LR[IdxSkids_LR].ErrorInfo.Text		:= 'ALARM_AB19.2';
				gSkid_LR[IdxSkids_LR].ErrorInfo.State		:= 'Warning';
				gSkid_LR[IdxSkids_LR].ErrorInfo.Severity	:= 1;
				gSkid_LR[IdxSkids_LR].Error := TRUE;
				gServices.Alarms_LR[IdxSkids_LR].Internal.Alarms_State.ALARM_AB19.2 := TRUE;
			END_IF
		END_IF;

		IF gSkid_LR[IdxSkids_LR].Alarms.ALARM_AB19.3 AND gServices.Alarms_LR[IdxSkids_LR].Internal.Alarms_State.ALARM_AB19.3 = FALSE THEN
			IF gSkid_LR[IdxSkids_LR].ErrorInfo.Text = '' THEN
				gSkid_LR[IdxSkids_LR].ErrorInfo.Text		:= 'ALARM_AB19.3';
				gSkid_LR[IdxSkids_LR].ErrorInfo.State		:= 'Warning';
				gSkid_LR[IdxSkids_LR].ErrorInfo.Severity	:= 1;
				gSkid_LR[IdxSkids_LR].Error := TRUE;
				gServices.Alarms_LR[IdxSkids_LR].Internal.Alarms_State.ALARM_AB19.3 := TRUE;
			END_IF
		END_IF;

		IF gSkid_LR[IdxSkids_LR].Alarms.ALARM_AB19.4 AND gServices.Alarms_LR[IdxSkids_LR].Internal.Alarms_State.ALARM_AB19.4 = FALSE THEN
			IF gSkid_LR[IdxSkids_LR].ErrorInfo.Text = '' THEN
				gSkid_LR[IdxSkids_LR].ErrorInfo.Text		:= 'ALARM_AB19.4';
				gSkid_LR[IdxSkids_LR].ErrorInfo.State		:= 'Warning';
				gSkid_LR[IdxSkids_LR].ErrorInfo.Severity	:= 1;
				gSkid_LR[IdxSkids_LR].Error := TRUE;
				gServices.Alarms_LR[IdxSkids_LR].Internal.Alarms_State.ALARM_AB19.4 := TRUE;
			END_IF
		END_IF;

		IF gSkid_LR[IdxSkids_LR].Alarms.ALARM_AB19.5 AND gServices.Alarms_LR[IdxSkids_LR].Internal.Alarms_State.ALARM_AB19.5 = FALSE THEN
			IF gSkid_LR[IdxSkids_LR].ErrorInfo.Text = '' THEN
				gSkid_LR[IdxSkids_LR].ErrorInfo.Text		:= 'ALARM_AB19.5';
				gSkid_LR[IdxSkids_LR].ErrorInfo.State		:= 'Warning';
				gSkid_LR[IdxSkids_LR].ErrorInfo.Severity	:= 1;
				gSkid_LR[IdxSkids_LR].Error := TRUE;
				gServices.Alarms_LR[IdxSkids_LR].Internal.Alarms_State.ALARM_AB19.5 := TRUE;
			END_IF
		END_IF;

		IF gSkid_LR[IdxSkids_LR].Alarms.ALARM_AB19.6 AND gServices.Alarms_LR[IdxSkids_LR].Internal.Alarms_State.ALARM_AB19.6 = FALSE THEN
			IF gSkid_LR[IdxSkids_LR].ErrorInfo.Text = '' THEN
				gSkid_LR[IdxSkids_LR].ErrorInfo.Text		:= 'ALARM_AB19.6';
				gSkid_LR[IdxSkids_LR].ErrorInfo.State		:= 'Warning';
				gSkid_LR[IdxSkids_LR].ErrorInfo.Severity	:= 1;
				gSkid_LR[IdxSkids_LR].Error := TRUE;
				gServices.Alarms_LR[IdxSkids_LR].Internal.Alarms_State.ALARM_AB19.6 := TRUE;
			END_IF
		END_IF;
		IF gSkid_LR[IdxSkids_LR].Alarms.ALARM_AB19.7 AND gServices.Alarms_LR[IdxSkids_LR].Internal.Alarms_State.ALARM_AB19.7 = FALSE THEN
			IF gSkid_LR[IdxSkids_LR].ErrorInfo.Text = '' THEN
				gSkid_LR[IdxSkids_LR].ErrorInfo.Text		:= 'ALARM_AB19.7';
				gSkid_LR[IdxSkids_LR].ErrorInfo.State		:= 'Warning';
				gSkid_LR[IdxSkids_LR].ErrorInfo.Severity	:= 1;
				gSkid_LR[IdxSkids_LR].Error := TRUE;
				gServices.Alarms_LR[IdxSkids_LR].Internal.Alarms_State.ALARM_AB19.7 := TRUE;
			END_IF
		END_IF;
		IF gSkid_LR[IdxSkids_LR].Alarms.ALARM_AB19.8 AND gServices.Alarms_LR[IdxSkids_LR].Internal.Alarms_State.ALARM_AB19.8 = FALSE THEN
			IF gSkid_LR[IdxSkids_LR].ErrorInfo.Text = '' THEN
				gSkid_LR[IdxSkids_LR].ErrorInfo.Text		:= 'ALARM_AB19.8';
				gSkid_LR[IdxSkids_LR].ErrorInfo.State		:= 'Warning';
				gSkid_LR[IdxSkids_LR].ErrorInfo.Severity	:= 1;
				gSkid_LR[IdxSkids_LR].Error := TRUE;
				gServices.Alarms_LR[IdxSkids_LR].Internal.Alarms_State.ALARM_AB19.8 := TRUE;
			END_IF
		END_IF;
		IF gSkid_LR[IdxSkids_LR].Alarms.ALARM_AB19.9 AND gServices.Alarms_LR[IdxSkids_LR].Internal.Alarms_State.ALARM_AB19.9 = FALSE THEN
			IF gSkid_LR[IdxSkids_LR].ErrorInfo.Text = '' THEN
				gSkid_LR[IdxSkids_LR].ErrorInfo.Text		:= 'ALARM_AB19.9';
				gSkid_LR[IdxSkids_LR].ErrorInfo.State		:= 'Warning';
				gSkid_LR[IdxSkids_LR].ErrorInfo.Severity	:= 1;
				gSkid_LR[IdxSkids_LR].Error := TRUE;
				gServices.Alarms_LR[IdxSkids_LR].Internal.Alarms_State.ALARM_AB19.9 := TRUE;
			END_IF
		END_IF;
		IF gSkid_LR[IdxSkids_LR].Alarms.ALARM_AB19.10 AND gServices.Alarms_LR[IdxSkids_LR].Internal.Alarms_State.ALARM_AB19.10 = FALSE THEN
			IF gSkid_LR[IdxSkids_LR].ErrorInfo.Text = '' THEN
				gSkid_LR[IdxSkids_LR].ErrorInfo.Text		:= 'ALARM_AB19.10';
				gSkid_LR[IdxSkids_LR].ErrorInfo.State		:= 'Warning';
				gSkid_LR[IdxSkids_LR].ErrorInfo.Severity	:= 1;
				gSkid_LR[IdxSkids_LR].Error := TRUE;
				gServices.Alarms_LR[IdxSkids_LR].Internal.Alarms_State.ALARM_AB19.10 := TRUE;
			END_IF
		END_IF;
		IF gSkid_LR[IdxSkids_LR].Alarms.ALARM_AB19.11 AND gServices.Alarms_LR[IdxSkids_LR].Internal.Alarms_State.ALARM_AB19.11 = FALSE THEN
			IF gSkid_LR[IdxSkids_LR].ErrorInfo.Text = '' THEN
				gSkid_LR[IdxSkids_LR].ErrorInfo.Text		:= 'ALARM_AB19.11';
				gSkid_LR[IdxSkids_LR].ErrorInfo.State		:= 'Warning';
				gSkid_LR[IdxSkids_LR].ErrorInfo.Severity	:= 1;
				gSkid_LR[IdxSkids_LR].Error := TRUE;
				gServices.Alarms_LR[IdxSkids_LR].Internal.Alarms_State.ALARM_AB19.11 := TRUE;
			END_IF
		END_IF;
		IF gSkid_LR[IdxSkids_LR].Alarms.ALARM_AB19.12 AND gServices.Alarms_LR[IdxSkids_LR].Internal.Alarms_State.ALARM_AB19.12 = FALSE THEN
			IF gSkid_LR[IdxSkids_LR].ErrorInfo.Text = '' THEN
				gSkid_LR[IdxSkids_LR].ErrorInfo.Text		:= 'ALARM_AB19.12';
				gSkid_LR[IdxSkids_LR].ErrorInfo.State		:= 'Warning';
				gSkid_LR[IdxSkids_LR].ErrorInfo.Severity	:= 1;
				gSkid_LR[IdxSkids_LR].Error := TRUE;
				gServices.Alarms_LR[IdxSkids_LR].Internal.Alarms_State.ALARM_AB19.12 := TRUE;
			END_IF
		END_IF;

	END_IF;

	(*********************************************************************Dont Touch This Code**********************************************************************)
	IF gSkid_LR[IdxSkids_LR].Error AND gSkid_LR[IdxSkids_LR].AlarmsInitialized AND gSkid_LR[IdxSkids_LR].Pmax_General_Variables.UNIT_ID <> 0 AND gUnit_LR[IdxSkids_LR] <> 0 THEN
		CASE gSkid_LR[IdxSkids_LR].ErrorInfo.Severity OF
			1:
				gSkid_LR[IdxSkids_LR].tempAlarm.name			:= 'Severity1';
				gSkid_LR[IdxSkids_LR].tempAlarm.allowMultiple	:= TRUE;
				gSkid_LR[IdxSkids_LR].tempAlarm.addText[0]		:= gSkid_LR[IdxSkids_LR].ErrorInfo.State;
				gSkid_LR[IdxSkids_LR].tempAlarm.addText[1]		:= gSkid_LR[IdxSkids_LR].ErrorInfo.Text;

				HA_Array_AddTop(ADR(gServices.Alarms_LR[IdxSkids_LR].In.AlarmList), SIZEOF(gServices.Alarms_LR[IdxSkids_LR].In.AlarmList), ADR(gSkid_LR[IdxSkids_LR].tempAlarm), SIZEOF(gSkid_LR[IdxSkids_LR].tempAlarm));

				gSkid_LR[IdxSkids_LR].tempAlarm.name			:= UINT_TO_STRING(gUnit_LR[IdxSkids_LR]);
				gSkid_LR[IdxSkids_LR].tempAlarm.name			:= CONCAT('Skid',gSkid_LR[IdxSkids_LR].tempAlarm.name);
				gSkid_LR[IdxSkids_LR].tempAlarm.name			:= CONCAT(gSkid_LR[IdxSkids_LR].tempAlarm.name,'Severity1');
				gSkid_LR[IdxSkids_LR].tempAlarm.allowMultiple	:= FALSE;
				gSkid_LR[IdxSkids_LR].tempAlarm.addText[1]		:= 'GENERAL_SEVERITY1';

				HA_Array_AddTop(ADR(gServices.Alarms_Global.AlarmList), SIZEOF(gServices.Alarms_Global.AlarmList), ADR(gSkid_LR[IdxSkids_LR].tempAlarm), SIZEOF(gSkid_LR[IdxSkids_LR].tempAlarm));

			2:
				gSkid_LR[IdxSkids_LR].tempAlarm.name			:= 'Severity2';
				gSkid_LR[IdxSkids_LR].tempAlarm.allowMultiple	:= TRUE;
				gSkid_LR[IdxSkids_LR].tempAlarm.addText[0]		:= gSkid_LR[IdxSkids_LR].ErrorInfo.State;
				gSkid_LR[IdxSkids_LR].tempAlarm.addText[1]		:= gSkid_LR[IdxSkids_LR].ErrorInfo.Text;

				HA_Array_AddTop(ADR(gServices.Alarms_LR[IdxSkids_LR].In.AlarmList), SIZEOF(gServices.Alarms_LR[IdxSkids_LR].In.AlarmList), ADR(gSkid_LR[IdxSkids_LR].tempAlarm), SIZEOF(gSkid_LR[IdxSkids_LR].tempAlarm));

				gSkid_LR[IdxSkids_LR].tempAlarm.name			:= UINT_TO_STRING(gUnit_LR[IdxSkids_LR]);
				gSkid_LR[IdxSkids_LR].tempAlarm.name			:= CONCAT('Skid',gSkid_LR[IdxSkids_LR].tempAlarm.name);
				gSkid_LR[IdxSkids_LR].tempAlarm.name			:= CONCAT(gSkid_LR[IdxSkids_LR].tempAlarm.name,'Severity2');
				gSkid_LR[IdxSkids_LR].tempAlarm.allowMultiple	:= FALSE;
				gSkid_LR[IdxSkids_LR].tempAlarm.addText[1]		:= 'GENERAL_SEVERITY2';

				HA_Array_AddTop(ADR(gServices.Alarms_Global.AlarmList), SIZEOF(gServices.Alarms_Global.AlarmList), ADR(gSkid_LR[IdxSkids_LR].tempAlarm), SIZEOF(gSkid_LR[IdxSkids_LR].tempAlarm));

			3:
				gSkid_LR[IdxSkids_LR].tempAlarm.name			:= 'Severity3';
				gSkid_LR[IdxSkids_LR].tempAlarm.allowMultiple	:= TRUE;
				gSkid_LR[IdxSkids_LR].tempAlarm.addText[0]		:= gSkid_LR[IdxSkids_LR].ErrorInfo.State;
				gSkid_LR[IdxSkids_LR].tempAlarm.addText[1]		:= gSkid_LR[IdxSkids_LR].ErrorInfo.Text;

				HA_Array_AddTop(ADR(gServices.Alarms_LR[IdxSkids_LR].In.AlarmList), SIZEOF(gServices.Alarms_LR[IdxSkids_LR].In.AlarmList), ADR(gSkid_LR[IdxSkids_LR].tempAlarm), SIZEOF(gSkid_LR[IdxSkids_LR].tempAlarm));

				gSkid_LR[IdxSkids_LR].tempAlarm.name			:= UINT_TO_STRING(gUnit_LR[IdxSkids_LR]);
				gSkid_LR[IdxSkids_LR].tempAlarm.name			:= CONCAT('Skid',gSkid_LR[IdxSkids_LR].tempAlarm.name);
				gSkid_LR[IdxSkids_LR].tempAlarm.name			:= CONCAT(gSkid_LR[IdxSkids_LR].tempAlarm.name,'Severity3');
				gSkid_LR[IdxSkids_LR].tempAlarm.allowMultiple	:= FALSE;
				gSkid_LR[IdxSkids_LR].tempAlarm.addText[1]		:= 'GENERAL_SEVERITY3';

				HA_Array_AddTop(ADR(gServices.Alarms_Global.AlarmList), SIZEOF(gServices.Alarms_Global.AlarmList), ADR(gSkid_LR[IdxSkids_LR].tempAlarm), SIZEOF(gSkid_LR[IdxSkids_LR].tempAlarm));

			4:
				gSkid_LR[IdxSkids_LR].tempAlarm.name			:= 'Severity4';
				gSkid_LR[IdxSkids_LR].tempAlarm.allowMultiple	:= TRUE;
				gSkid_LR[IdxSkids_LR].tempAlarm.addText[0]		:= gSkid_LR[IdxSkids_LR].ErrorInfo.State;
				gSkid_LR[IdxSkids_LR].tempAlarm.addText[1]		:= gSkid_LR[IdxSkids_LR].ErrorInfo.Text;

				HA_Array_AddTop(ADR(gServices.Alarms_LR[IdxSkids_LR].In.AlarmList), SIZEOF(gServices.Alarms_LR[IdxSkids_LR].In.AlarmList), ADR(gSkid_LR[IdxSkids_LR].tempAlarm), SIZEOF(gSkid_LR[IdxSkids_LR].tempAlarm));

				gSkid_LR[IdxSkids_LR].tempAlarm.name			:= UINT_TO_STRING(gUnit_LR[IdxSkids_LR]);
				gSkid_LR[IdxSkids_LR].tempAlarm.name			:= CONCAT('Skid',gSkid_LR[IdxSkids_LR].tempAlarm.name);
				gSkid_LR[IdxSkids_LR].tempAlarm.name			:= CONCAT(gSkid_LR[IdxSkids_LR].tempAlarm.name,'Severity4');
				gSkid_LR[IdxSkids_LR].tempAlarm.allowMultiple	:= FALSE;
				gSkid_LR[IdxSkids_LR].tempAlarm.addText[1]		:= 'GENERAL_SEVERITY4';

				HA_Array_AddTop(ADR(gServices.Alarms_Global.AlarmList), SIZEOF(gServices.Alarms_Global.AlarmList), ADR(gSkid_LR[IdxSkids_LR].tempAlarm), SIZEOF(gSkid_LR[IdxSkids_LR].tempAlarm));

			5:
				gSkid_LR[IdxSkids_LR].tempAlarm.name			:= 'Severity5';
				gSkid_LR[IdxSkids_LR].tempAlarm.allowMultiple	:= TRUE;
				gSkid_LR[IdxSkids_LR].tempAlarm.addText[0]		:= gSkid_LR[IdxSkids_LR].ErrorInfo.State;
				gSkid_LR[IdxSkids_LR].tempAlarm.addText[1]		:= gSkid_LR[IdxSkids_LR].ErrorInfo.Text;

				HA_Array_AddTop(ADR(gServices.Alarms_LR[IdxSkids_LR].In.AlarmList), SIZEOF(gServices.Alarms_LR[IdxSkids_LR].In.AlarmList), ADR(gSkid_LR[IdxSkids_LR].tempAlarm), SIZEOF(gSkid_LR[IdxSkids_LR].tempAlarm));

				gSkid_LR[IdxSkids_LR].tempAlarm.name			:= UINT_TO_STRING(gUnit_LR[IdxSkids_LR]);
				gSkid_LR[IdxSkids_LR].tempAlarm.name			:= CONCAT('Skid',gSkid_LR[IdxSkids_LR].tempAlarm.name);
				gSkid_LR[IdxSkids_LR].tempAlarm.name			:= CONCAT(gSkid_LR[IdxSkids_LR].tempAlarm.name,'Severity5');
				gSkid_LR[IdxSkids_LR].tempAlarm.allowMultiple	:= FALSE;
				gSkid_LR[IdxSkids_LR].tempAlarm.addText[1]		:= 'GENERAL_SEVERITY5';

				HA_Array_AddTop(ADR(gServices.Alarms_Global.AlarmList), SIZEOF(gServices.Alarms_Global.AlarmList), ADR(gSkid_LR[IdxSkids_LR].tempAlarm), SIZEOF(gSkid_LR[IdxSkids_LR].tempAlarm));

		END_CASE
		brsmemset(ADR(gSkid_LR[IdxSkids_LR].tempAlarm),0,SIZEOF(gSkid_LR[IdxSkids_LR].tempAlarm));
		gSkid_LR[IdxSkids_LR].Error := FALSE;

	END_IF

	brsmemset(ADR(gSkid_LR[IdxSkids_LR].ErrorInfo),0,SIZEOF(gSkid_LR[IdxSkids_LR].ErrorInfo));

	// Case for handling the alarm history
	CASE gServices.Alarms_LR[IdxSkids_LR].Internal.StateExportHistory OF
		0:
			IF gServices.Alarms_LR[IdxSkids_LR].In.ExportHistory THEN
				HA_AlarmX_Helper(gSkid_LR[IdxSkids_LR].AlarmX_MpLink,'',HA_ALARMX_ACTION_LOG_ONLY,'HISTORY EXPORTED',FALSE);
				gServices.Alarms_LR[IdxSkids_LR].In.ExportHistory 									:= FALSE;
				gServices.Alarms_LR[IdxSkids_LR].Internal.MpAlarmXHistory_0.Export 				:= TRUE;
				gServices.Alarms_LR[IdxSkids_LR].Internal.StateExportHistory 						:= 10;
			ELSIF gServices.Alarms_LR[IdxSkids_LR].In.ClearHistory THEN
				HA_AlarmX_Helper(gSkid_LR[IdxSkids_LR].AlarmX_MpLink,'',HA_ALARMX_ACTION_LOG_ONLY,'HISTORY CLEARED',FALSE);
				gServices.Alarms_LR[IdxSkids_LR].In.ClearHistory 									:= FALSE;
				MpAlarmXClearHistory(gSkid_LR[IdxSkids_LR].AlarmXHistory_MpLink);
			END_IF;
		10:
			IF gServices.Alarms_LR[IdxSkids_LR].Internal.MpAlarmXHistory_0.CommandDone OR gServices.Alarms_LR[IdxSkids_LR].Internal.MpAlarmXHistory_0.Error THEN
				gServices.Alarms_LR[IdxSkids_LR].Internal.MpAlarmXHistory_0.Export 				:= FALSE;
				gServices.Alarms_LR[IdxSkids_LR].Internal.StateExportHistory 						:= 0;
			END_IF;
	END_CASE;

	//	IF gMain.ErrorReset THEN
	//		gServices.Alarms_LR[IdxSkids_LR].In.ResetAlarms 											:= TRUE;
	//	END_IF;

	// Case for handling the alarm resetting
	CASE gServices.Alarms_LR[IdxSkids_LR].Internal.StateResetAlarms OF
		0:
			IF gServices.Alarms_LR[IdxSkids_LR].In.ResetAlarms OR gVis.Global.ErrorReset THEN
				HA_AlarmX_Helper(gSkid_LR[IdxSkids_LR].AlarmX_MpLink,'',HA_ALARMX_ACTION_LOG_ONLY,'ACKNOWLEDGE ALL',FALSE);
				gServices.Alarms_LR[IdxSkids_LR].In.ResetAlarms 									:= FALSE;
				gVis.Alarms_LR[IdxSkids_LR].Active.UIConnect.AcknowledgeAll 							:= TRUE;
				gServices.Alarms_LR[IdxSkids_LR].Internal.CTON_ResetDelay(IN := FALSE);
				gServices.Alarms_LR[IdxSkids_LR].Internal.StateResetAlarms 						:= 10;
			END_IF;
		10:
			// give UI time to process the reset
			IF gServices.Alarms_LR[IdxSkids_LR].Internal.CTON_ResetDelay.Q THEN
				gServices.Alarms_LR[IdxSkids_LR].Internal.CTON_ResetDelay(IN := FALSE);
				gServices.Alarms_LR[IdxSkids_LR].Internal.StateResetAlarms 						:= 0;
				gVis.Global.ErrorReset := FALSE;
			ELSE
				gServices.Alarms_LR[IdxSkids_LR].Internal.CTON_ResetDelay(IN := TRUE, PT := T#250ms);
			END_IF;
	END_CASE;

	//	//Set Unit Number and Add Alarms
	IF (gSkid_LR[IdxSkids_LR].Pmax_General_Variables.UNIT_ID <> 0 AND (gUnit_LR[IdxSkids_LR] <> gSkid_LR[IdxSkids_LR].Pmax_General_Variables.UNIT_ID))  THEN

		gUnit_LR[IdxSkids_LR] := gSkid_LR[IdxSkids_LR].Pmax_General_Variables.UNIT_ID;

		gSkid_LR[IdxSkids_LR].AlarmName	 := UINT_TO_STRING(gUnit_LR[IdxSkids_LR]);
		gSkid_LR[IdxSkids_LR].AlarmName	 := CONCAT('Skid',gSkid_LR[IdxSkids_LR].AlarmName	);

		gSkid_LR[IdxSkids_LR].i := 1;

		SkidNumberINT := UINT_TO_STRING(gUnit_LR[IdxSkids_LR]);

	END_IF;

	//Create Alarms
	CASE gSkid_LR[IdxSkids_LR].i OF
		0:
			//IDLE
		1:
			gSkid_LR[IdxSkids_LR].AlarmName	 := UINT_TO_STRING(gUnit_LR[IdxSkids_LR]);
			gSkid_LR[IdxSkids_LR].AlarmName	 := CONCAT('Skid',gSkid_LR[IdxSkids_LR].AlarmName	);
			HA_brsstrcat(ADR(gSkid_LR[IdxSkids_LR].AlarmName), ADR('Severity1'), SIZEOF(gSkid_LR[IdxSkids_LR].AlarmName));
			gSkid_LR[IdxSkids_LR].AlarmCfg.Message												:= '{$$IAT/GlobalAlarm.';
			HA_brsstrcat(ADR(gSkid_LR[IdxSkids_LR].AlarmCfg.Message), ADR('Severity1'), SIZEOF(gSkid_LR[IdxSkids_LR].AlarmCfg.Message));
			HA_brsstrcat(ADR(gSkid_LR[IdxSkids_LR].AlarmCfg.Message), ADR('}'), SIZEOF(gSkid_LR[IdxSkids_LR].AlarmCfg.Message));
			gSkid_LR[IdxSkids_LR].AlarmCfg.Code													:= gUnit_LR[IdxSkids_LR];
			gSkid_LR[IdxSkids_LR].AlarmCfg.Severity												:= 1;
			gSkid_LR[IdxSkids_LR].AlarmCfg.Behavior.AutoReset									:= TRUE;
			gSkid_LR[IdxSkids_LR].AlarmCfg.Behavior.Acknowledge 									:= mpALARMX_ACK_REQ;
			gSkid_LR[IdxSkids_LR].AlarmCfg.Behavior.MultipleInstances 							:= TRUE;
			gSkid_LR[IdxSkids_LR].AlarmCfg.Behavior.ReactionUntilAcknowledged					:= TRUE;
			gSkid_LR[IdxSkids_LR].AlarmCfg.Behavior.HistoryReport.AcknowledgedToUnacknowledged := FALSE;
			gSkid_LR[IdxSkids_LR].AlarmCfg.Behavior.HistoryReport.ActiveToInactive := FALSE;
			gSkid_LR[IdxSkids_LR].AlarmCfg.Behavior.HistoryReport.InactiveToActive := TRUE;
			gSkid_LR[IdxSkids_LR].AlarmCfg.Behavior.HistoryReport.Reactivation := FALSE;
			gSkid_LR[IdxSkids_LR].AlarmCfg.Behavior.HistoryReport.UnacknowledgedToAcknowledged := FALSE;
			gSkid_LR[IdxSkids_LR].MpAlarmXConfigAlarm.Save				:= TRUE;

		2:
			gSkid_LR[IdxSkids_LR].AlarmName	 := UINT_TO_STRING(gUnit_LR[IdxSkids_LR]);
			gSkid_LR[IdxSkids_LR].AlarmName	 := CONCAT('Skid',gSkid_LR[IdxSkids_LR].AlarmName	);
			HA_brsstrcat(ADR(gSkid_LR[IdxSkids_LR].AlarmName), ADR('Severity2'), SIZEOF(gSkid_LR[IdxSkids_LR].AlarmName));
			gSkid_LR[IdxSkids_LR].AlarmCfg.Message												:= '{$$IAT/GlobalAlarm.';
			HA_brsstrcat(ADR(gSkid_LR[IdxSkids_LR].AlarmCfg.Message), ADR('Severity2'), SIZEOF(gSkid_LR[IdxSkids_LR].AlarmCfg.Message));
			HA_brsstrcat(ADR(gSkid_LR[IdxSkids_LR].AlarmCfg.Message), ADR('}'), SIZEOF(gSkid_LR[IdxSkids_LR].AlarmCfg.Message));
			gSkid_LR[IdxSkids_LR].AlarmCfg.Code													:= gUnit_LR[IdxSkids_LR];
			gSkid_LR[IdxSkids_LR].AlarmCfg.Severity												:= 2;
			gSkid_LR[IdxSkids_LR].AlarmCfg.Behavior.AutoReset									:= TRUE;
			gSkid_LR[IdxSkids_LR].AlarmCfg.Behavior.Acknowledge 									:= mpALARMX_ACK_REQ;
			gSkid_LR[IdxSkids_LR].AlarmCfg.Behavior.MultipleInstances 							:= TRUE;
			gSkid_LR[IdxSkids_LR].AlarmCfg.Behavior.ReactionUntilAcknowledged					:= TRUE;
			gSkid_LR[IdxSkids_LR].AlarmCfg.Behavior.HistoryReport.AcknowledgedToUnacknowledged := FALSE;
			gSkid_LR[IdxSkids_LR].AlarmCfg.Behavior.HistoryReport.ActiveToInactive := FALSE;
			gSkid_LR[IdxSkids_LR].AlarmCfg.Behavior.HistoryReport.InactiveToActive := TRUE;
			gSkid_LR[IdxSkids_LR].AlarmCfg.Behavior.HistoryReport.Reactivation := FALSE;
			gSkid_LR[IdxSkids_LR].AlarmCfg.Behavior.HistoryReport.UnacknowledgedToAcknowledged := FALSE;
			gSkid_LR[IdxSkids_LR].MpAlarmXConfigAlarm.Save				:= TRUE;

		3:
			gSkid_LR[IdxSkids_LR].AlarmName	 := UINT_TO_STRING(gUnit_LR[IdxSkids_LR]);
			gSkid_LR[IdxSkids_LR].AlarmName	 := CONCAT('Skid',gSkid_LR[IdxSkids_LR].AlarmName	);
			HA_brsstrcat(ADR(gSkid_LR[IdxSkids_LR].AlarmName), ADR('Severity3'), SIZEOF(gSkid_LR[IdxSkids_LR].AlarmName));
			gSkid_LR[IdxSkids_LR].AlarmCfg.Message												:= '{$$IAT/GlobalAlarm.';
			HA_brsstrcat(ADR(gSkid_LR[IdxSkids_LR].AlarmCfg.Message), ADR('Severity3'), SIZEOF(gSkid_LR[IdxSkids_LR].AlarmCfg.Message));
			HA_brsstrcat(ADR(gSkid_LR[IdxSkids_LR].AlarmCfg.Message), ADR('}'), SIZEOF(gSkid_LR[IdxSkids_LR].AlarmCfg.Message));
			gSkid_LR[IdxSkids_LR].AlarmCfg.Code													:= gUnit_LR[IdxSkids_LR];
			gSkid_LR[IdxSkids_LR].AlarmCfg.Severity												:= 3;
			gSkid_LR[IdxSkids_LR].AlarmCfg.Behavior.AutoReset									:= TRUE;
			gSkid_LR[IdxSkids_LR].AlarmCfg.Behavior.Acknowledge 									:= mpALARMX_ACK_REQ;
			gSkid_LR[IdxSkids_LR].AlarmCfg.Behavior.MultipleInstances 							:= TRUE;
			gSkid_LR[IdxSkids_LR].AlarmCfg.Behavior.ReactionUntilAcknowledged					:= TRUE;
			gSkid_LR[IdxSkids_LR].AlarmCfg.Behavior.HistoryReport.AcknowledgedToUnacknowledged := FALSE;
			gSkid_LR[IdxSkids_LR].AlarmCfg.Behavior.HistoryReport.ActiveToInactive := FALSE;
			gSkid_LR[IdxSkids_LR].AlarmCfg.Behavior.HistoryReport.InactiveToActive := TRUE;
			gSkid_LR[IdxSkids_LR].AlarmCfg.Behavior.HistoryReport.Reactivation := FALSE;
			gSkid_LR[IdxSkids_LR].AlarmCfg.Behavior.HistoryReport.UnacknowledgedToAcknowledged := FALSE;
			gSkid_LR[IdxSkids_LR].MpAlarmXConfigAlarm.Save				:= TRUE;

		4:
			gSkid_LR[IdxSkids_LR].AlarmName	 := UINT_TO_STRING(gUnit_LR[IdxSkids_LR]);
			gSkid_LR[IdxSkids_LR].AlarmName	 := CONCAT('Skid',gSkid_LR[IdxSkids_LR].AlarmName	);
			HA_brsstrcat(ADR(gSkid_LR[IdxSkids_LR].AlarmName), ADR('Severity4'), SIZEOF(gSkid_LR[IdxSkids_LR].AlarmName));
			gSkid_LR[IdxSkids_LR].AlarmCfg.Message												:= '{$$IAT/GlobalAlarm.';
			HA_brsstrcat(ADR(gSkid_LR[IdxSkids_LR].AlarmCfg.Message), ADR('Severity4'), SIZEOF(gSkid_LR[IdxSkids_LR].AlarmCfg.Message));
			HA_brsstrcat(ADR(gSkid_LR[IdxSkids_LR].AlarmCfg.Message), ADR('}'), SIZEOF(gSkid_LR[IdxSkids_LR].AlarmCfg.Message));
			gSkid_LR[IdxSkids_LR].AlarmCfg.Code													:= gUnit_LR[IdxSkids_LR];
			gSkid_LR[IdxSkids_LR].AlarmCfg.Severity												:= 4;
			gSkid_LR[IdxSkids_LR].AlarmCfg.Behavior.AutoReset									:= TRUE;
			gSkid_LR[IdxSkids_LR].AlarmCfg.Behavior.Acknowledge 									:= mpALARMX_ACK_REQ;
			gSkid_LR[IdxSkids_LR].AlarmCfg.Behavior.MultipleInstances 							:= TRUE;
			gSkid_LR[IdxSkids_LR].AlarmCfg.Behavior.ReactionUntilAcknowledged					:= TRUE;
			gSkid_LR[IdxSkids_LR].AlarmCfg.Behavior.HistoryReport.AcknowledgedToUnacknowledged := FALSE;
			gSkid_LR[IdxSkids_LR].AlarmCfg.Behavior.HistoryReport.ActiveToInactive := FALSE;
			gSkid_LR[IdxSkids_LR].AlarmCfg.Behavior.HistoryReport.InactiveToActive := TRUE;
			gSkid_LR[IdxSkids_LR].AlarmCfg.Behavior.HistoryReport.Reactivation := FALSE;
			gSkid_LR[IdxSkids_LR].AlarmCfg.Behavior.HistoryReport.UnacknowledgedToAcknowledged := FALSE;
			gSkid_LR[IdxSkids_LR].MpAlarmXConfigAlarm.Save				:= TRUE;
		5:
			gSkid_LR[IdxSkids_LR].AlarmName	 := UINT_TO_STRING(gUnit_LR[IdxSkids_LR]);
			gSkid_LR[IdxSkids_LR].AlarmName	 := CONCAT('Skid',gSkid_LR[IdxSkids_LR].AlarmName	);
			HA_brsstrcat(ADR(gSkid_LR[IdxSkids_LR].AlarmName), ADR('Severity5'), SIZEOF(gSkid_LR[IdxSkids_LR].AlarmName));
			gSkid_LR[IdxSkids_LR].AlarmCfg.Message												:= '{$$IAT/GlobalAlarm.';
			HA_brsstrcat(ADR(gSkid_LR[IdxSkids_LR].AlarmCfg.Message), ADR('Severity5'), SIZEOF(gSkid_LR[IdxSkids_LR].AlarmCfg.Message));
			HA_brsstrcat(ADR(gSkid_LR[IdxSkids_LR].AlarmCfg.Message), ADR('}'), SIZEOF(gSkid_LR[IdxSkids_LR].AlarmCfg.Message));
			gSkid_LR[IdxSkids_LR].AlarmCfg.Code													:= gUnit_LR[IdxSkids_LR];
			gSkid_LR[IdxSkids_LR].AlarmCfg.Severity												:= 5;
			gSkid_LR[IdxSkids_LR].AlarmCfg.Behavior.AutoReset									:= TRUE;
			gSkid_LR[IdxSkids_LR].AlarmCfg.Behavior.Acknowledge 									:= mpALARMX_ACK_REQ;
			gSkid_LR[IdxSkids_LR].AlarmCfg.Behavior.MultipleInstances 							:= TRUE;
			gSkid_LR[IdxSkids_LR].AlarmCfg.Behavior.ReactionUntilAcknowledged					:= TRUE;
			gSkid_LR[IdxSkids_LR].AlarmCfg.Behavior.HistoryReport.AcknowledgedToUnacknowledged := FALSE;
			gSkid_LR[IdxSkids_LR].AlarmCfg.Behavior.HistoryReport.ActiveToInactive := FALSE;
			gSkid_LR[IdxSkids_LR].AlarmCfg.Behavior.HistoryReport.InactiveToActive := TRUE;
			gSkid_LR[IdxSkids_LR].AlarmCfg.Behavior.HistoryReport.Reactivation := FALSE;
			gSkid_LR[IdxSkids_LR].AlarmCfg.Behavior.HistoryReport.UnacknowledgedToAcknowledged := FALSE;
			gSkid_LR[IdxSkids_LR].MpAlarmXConfigAlarm.Save				:= TRUE;

		6:
			gSkid_LR[IdxSkids_LR].AlarmName	 := UINT_TO_STRING(gUnit_LR[IdxSkids_LR]);
			gSkid_LR[IdxSkids_LR].AlarmName	 := CONCAT('Skid',gSkid_LR[IdxSkids_LR].AlarmName	);
			HA_brsstrcat(ADR(gSkid_LR[IdxSkids_LR].AlarmName), ADR('CmdIgnored'), SIZEOF(gSkid_LR[IdxSkids_LR].AlarmName));
			gSkid_LR[IdxSkids_LR].AlarmCfg.Message												:= '{$$IAT/GlobalAlarm.';
			HA_brsstrcat(ADR(gSkid_LR[IdxSkids_LR].AlarmCfg.Message), ADR(gSkid_LR[IdxSkids_LR].AlarmName), SIZEOF(gSkid_LR[IdxSkids_LR].AlarmCfg.Message));
			HA_brsstrcat(ADR(gSkid_LR[IdxSkids_LR].AlarmCfg.Message), ADR('}'), SIZEOF(gSkid_LR[IdxSkids_LR].AlarmCfg.Message));
			gSkid_LR[IdxSkids_LR].AlarmCfg.Code													:= gUnit_LR[IdxSkids_LR] + 6;
			gSkid_LR[IdxSkids_LR].AlarmCfg.Severity												:= 0;
			gSkid_LR[IdxSkids_LR].AlarmCfg.Behavior.AutoReset									:= TRUE;
			gSkid_LR[IdxSkids_LR].AlarmCfg.Behavior.Acknowledge 									:= mpALARMX_ACK_REQ;
			gSkid_LR[IdxSkids_LR].AlarmCfg.Behavior.MultipleInstances 							:= TRUE;
			gSkid_LR[IdxSkids_LR].AlarmCfg.Behavior.ReactionUntilAcknowledged					:= TRUE;
			gSkid_LR[IdxSkids_LR].AlarmCfg.Behavior.HistoryReport.AcknowledgedToUnacknowledged := FALSE;
			gSkid_LR[IdxSkids_LR].AlarmCfg.Behavior.HistoryReport.ActiveToInactive := FALSE;
			gSkid_LR[IdxSkids_LR].AlarmCfg.Behavior.HistoryReport.InactiveToActive := TRUE;
			gSkid_LR[IdxSkids_LR].AlarmCfg.Behavior.HistoryReport.Reactivation := FALSE;
			gSkid_LR[IdxSkids_LR].AlarmCfg.Behavior.HistoryReport.UnacknowledgedToAcknowledged := FALSE;
			gSkid_LR[IdxSkids_LR].MpAlarmXConfigAlarm.Save				:= TRUE;
		7:
			gSkid_LR[IdxSkids_LR].AlarmStartupDelay.IN := TRUE;

			IF 	gSkid_LR[IdxSkids_LR].AlarmStartupDelay.Q THEN
				gSkid_LR[IdxSkids_LR].AlarmsInitialized := TRUE;
			END_IF;

	END_CASE

	gSkid_LR[IdxSkids_LR].AlarmStartupDelay(PT := T#30s);

	gSkid_LR[IdxSkids_LR].MpAlarmXConfigAlarm.MpLink			:= ADR(gAlarmXCore_Global);
	gSkid_LR[IdxSkids_LR].MpAlarmXConfigAlarm.Enable			:= TRUE;
	gSkid_LR[IdxSkids_LR].MpAlarmXConfigAlarm.Name				:= ADR(gSkid_LR[IdxSkids_LR].AlarmName);
	gSkid_LR[IdxSkids_LR].MpAlarmXConfigAlarm.Configuration	:= ADR(gSkid_LR[IdxSkids_LR].AlarmCfg);

	IF gSkid_LR[IdxSkids_LR].MpAlarmXConfigAlarm.CommandDone THEN
		IF gSkid_LR[IdxSkids_LR].i < 7 THEN
			gSkid_LR[IdxSkids_LR].i := gSkid_LR[IdxSkids_LR].i + 1;
		ELSE
			//Do nothing
		END_IF;

		gSkid_LR[IdxSkids_LR].MpAlarmXConfigAlarm.Save := FALSE;
	END_IF;

	gSkid_LR[IdxSkids_LR].MpAlarmXConfigAlarm();

END_ACTION
```

#### CMD.st
```iecst
ACTION Modbus_CMD_action:

	// --------------------------------------------------------------------
	// Variable Write Commands
	// --------------------------------------------------------------------

	// AS Block 12 - UNIT_ID
	IF gCMD_LR[IdxSkids_LR].Write_UNIT_ID.Send THEN
		MasterConfig_LR[IdxSkids_LR].action_enable[11].single := TRUE;
		gCMD_LR[IdxSkids_LR].Write_UNIT_ID.Send := FALSE;
	END_IF;

	// AS Block 13 - P201_STRT_CMD
	IF gCMD_LR[IdxSkids_LR].Write_P201_STRT_CMD.Send THEN
		MasterConfig_LR[IdxSkids_LR].action_enable[12].single := TRUE;
		gCMD_LR[IdxSkids_LR].Write_P201_STRT_CMD.Send := FALSE;
	END_IF;

	// AS Block 14 - P201_STP_CMD
	IF gCMD_LR[IdxSkids_LR].Write_P201_STP_CMD.Send THEN
		MasterConfig_LR[IdxSkids_LR].action_enable[13].single := TRUE;
		gCMD_LR[IdxSkids_LR].Write_P201_STP_CMD.Send := FALSE;
	END_IF;

	// AS Block 15 - P201_HOA
	IF gCMD_LR[IdxSkids_LR].Write_P201_HOA.Send THEN
		gCMD_LR[IdxSkids_LR].Write_P201_HOA.wP201_HOA := STRING_TO_UINT(gCMD_LR[IdxSkids_LR].Write_P201_HOA.wP201_HOA_String);
		MasterConfig_LR[IdxSkids_LR].action_enable[14].single := TRUE;
		gCMD_LR[IdxSkids_LR].Write_P201_HOA.Send := FALSE;
	ELSIF NOT gVis.Main.Out.DialogOpen THEN
		gCMD_LR[IdxSkids_LR].Write_P201_HOA.wP201_HOA_String := UINT_TO_STRING(gSkid_LR[IdxSkids_LR].Dosing_Pump_201.P201_HOA);
	END_IF;

	// AS Block 16 - P201_PPM
	IF gCMD_LR[IdxSkids_LR].Write_P201_PPM.Send THEN
		gCMD_LR[IdxSkids_LR].Write_P201_PPM.wP201_PPM_SWAPPED := IDEC_REAL_Conv(gCMD_LR[IdxSkids_LR].Write_P201_PPM.wP201_PPM);
		MasterConfig_LR[IdxSkids_LR].action_enable[15].single := TRUE;
		gCMD_LR[IdxSkids_LR].Write_P201_PPM.Send := FALSE;
	END_IF;

	// AS Block 17 - P201_SP
	IF gCMD_LR[IdxSkids_LR].Write_P201_SP.Send THEN
		gCMD_LR[IdxSkids_LR].Write_P201_SP.wP201_SP_SWAPPED := IDEC_REAL_Conv(gCMD_LR[IdxSkids_LR].Write_P201_SP.wP201_SP);
		MasterConfig_LR[IdxSkids_LR].action_enable[16].single := TRUE;
		gCMD_LR[IdxSkids_LR].Write_P201_SP.Send := FALSE;
	END_IF;

	// AS Block 18 - P202_STRT_CMD
	IF gCMD_LR[IdxSkids_LR].Write_P202_STRT_CMD.Send THEN
		MasterConfig_LR[IdxSkids_LR].action_enable[17].single := TRUE;
		gCMD_LR[IdxSkids_LR].Write_P202_STRT_CMD.Send := FALSE;
	END_IF;

	// AS Block 19 - P202_STP_CMD
	IF gCMD_LR[IdxSkids_LR].Write_P202_STP_CMD.Send THEN
		MasterConfig_LR[IdxSkids_LR].action_enable[18].single := TRUE;
		gCMD_LR[IdxSkids_LR].Write_P202_STP_CMD.Send := FALSE;
	END_IF;

	// AS Block 20 - P202_HOA
	IF gCMD_LR[IdxSkids_LR].Write_P202_HOA.Send THEN
		gCMD_LR[IdxSkids_LR].Write_P202_HOA.wP202_HOA := STRING_TO_UINT(gCMD_LR[IdxSkids_LR].Write_P202_HOA.wP202_HOA_String);
		MasterConfig_LR[IdxSkids_LR].action_enable[19].single := TRUE;
		gCMD_LR[IdxSkids_LR].Write_P202_HOA.Send := FALSE;
	ELSIF NOT gVis.Main.Out.DialogOpen THEN
		gCMD_LR[IdxSkids_LR].Write_P202_HOA.wP202_HOA_String := UINT_TO_STRING(gSkid_LR[IdxSkids_LR].Dosing_Pump_202.P202_HOA);
	END_IF;

	// AS Block 21 - P202_PPM
	IF gCMD_LR[IdxSkids_LR].Write_P202_PPM.Send THEN
		gCMD_LR[IdxSkids_LR].Write_P202_PPM.wP202_PPM_SWAPPED := IDEC_REAL_Conv(gCMD_LR[IdxSkids_LR].Write_P202_PPM.wP202_PPM);
		MasterConfig_LR[IdxSkids_LR].action_enable[20].single := TRUE;
		gCMD_LR[IdxSkids_LR].Write_P202_PPM.Send := FALSE;
	END_IF;

	// AS Block 22 - P202_SP
	IF gCMD_LR[IdxSkids_LR].Write_P202_SP.Send THEN
		gCMD_LR[IdxSkids_LR].Write_P202_SP.wP202_SP_SWAPPED := IDEC_REAL_Conv(gCMD_LR[IdxSkids_LR].Write_P202_SP.wP202_SP);
		MasterConfig_LR[IdxSkids_LR].action_enable[21].single := TRUE;
		gCMD_LR[IdxSkids_LR].Write_P202_SP.Send := FALSE;
	END_IF;

	// AS Block 23 - P203_STRT_CMD
	IF gCMD_LR[IdxSkids_LR].Write_P203_STRT_CMD.Send THEN
		MasterConfig_LR[IdxSkids_LR].action_enable[22].single := TRUE;
		gCMD_LR[IdxSkids_LR].Write_P203_STRT_CMD.Send := FALSE;
	END_IF;

	// AS Block 24 - P203_STP_CMD
	IF gCMD_LR[IdxSkids_LR].Write_P203_STP_CMD.Send THEN
		MasterConfig_LR[IdxSkids_LR].action_enable[23].single := TRUE;
		gCMD_LR[IdxSkids_LR].Write_P203_STP_CMD.Send := FALSE;
	END_IF;

	// AS Block 25 - P203_HOA
	IF gCMD_LR[IdxSkids_LR].Write_P203_HOA.Send THEN
		gCMD_LR[IdxSkids_LR].Write_P203_HOA.wP203_HOA := STRING_TO_UINT(gCMD_LR[IdxSkids_LR].Write_P203_HOA.wP203_HOA_String);
		MasterConfig_LR[IdxSkids_LR].action_enable[24].single := TRUE;
		gCMD_LR[IdxSkids_LR].Write_P203_HOA.Send := FALSE;
	ELSIF NOT gVis.Main.Out.DialogOpen THEN
		gCMD_LR[IdxSkids_LR].Write_P203_HOA.wP203_HOA_String := UINT_TO_STRING(gSkid_LR[IdxSkids_LR].Dosing_Pump_203.P203_HOA);
	END_IF;

	// AS Block 26 - P203_PPM
	IF gCMD_LR[IdxSkids_LR].Write_P203_PPM.Send THEN
		gCMD_LR[IdxSkids_LR].Write_P203_PPM.wP203_PPM_SWAPPED := IDEC_REAL_Conv(gCMD_LR[IdxSkids_LR].Write_P203_PPM.wP203_PPM);
		MasterConfig_LR[IdxSkids_LR].action_enable[25].single := TRUE;
		gCMD_LR[IdxSkids_LR].Write_P203_PPM.Send := FALSE;
	END_IF;

	// AS Block 27 - P203_SP
	IF gCMD_LR[IdxSkids_LR].Write_P203_SP.Send THEN
		gCMD_LR[IdxSkids_LR].Write_P203_SP.wP203_SP_SWAPPED := IDEC_REAL_Conv(gCMD_LR[IdxSkids_LR].Write_P203_SP.wP203_SP);
		MasterConfig_LR[IdxSkids_LR].action_enable[26].single := TRUE;
		gCMD_LR[IdxSkids_LR].Write_P203_SP.Send := FALSE;
	END_IF;

	// AS Block 28 - EFF_1
	IF gCMD_LR[IdxSkids_LR].Write_EFF_1.Send THEN
		gCMD_LR[IdxSkids_LR].Write_EFF_1.wEFF_1_SWAPPED := IDEC_REAL_Conv(gCMD_LR[IdxSkids_LR].Write_EFF_1.wEFF_1);
		MasterConfig_LR[IdxSkids_LR].action_enable[27].single := TRUE;
		MasterConfig_LR[IdxSkids_LR].action_enable[71].single := TRUE; // Send Recalculation Command
		gCMD_LR[IdxSkids_LR].Write_EFF_1.Send := FALSE;
	END_IF;

	// AS Block 29 - EFF_2
	IF gCMD_LR[IdxSkids_LR].Write_EFF_2.Send THEN
		gCMD_LR[IdxSkids_LR].Write_EFF_2.wEFF_2_SWAPPED := IDEC_REAL_Conv(gCMD_LR[IdxSkids_LR].Write_EFF_2.wEFF_2);
		MasterConfig_LR[IdxSkids_LR].action_enable[28].single := TRUE;
		MasterConfig_LR[IdxSkids_LR].action_enable[71].single := TRUE; // Send Recalculation Command
		gCMD_LR[IdxSkids_LR].Write_EFF_2.Send := FALSE;
	END_IF;

	// AS Block 30 - NAOH_TO_H2O2
	IF gCMD_LR[IdxSkids_LR].Write_NAOH_TO_H2O2.Send THEN
		gCMD_LR[IdxSkids_LR].Write_NAOH_TO_H2O2.wNAOH_TO_H2O2_SWAPPED := IDEC_REAL_Conv(gCMD_LR[IdxSkids_LR].Write_NAOH_TO_H2O2.wNAOH_TO_H2O2);
		MasterConfig_LR[IdxSkids_LR].action_enable[29].single := TRUE;
		MasterConfig_LR[IdxSkids_LR].action_enable[71].single := TRUE; // Send Recalculation Command
		gCMD_LR[IdxSkids_LR].Write_NAOH_TO_H2O2.Send := FALSE;
	END_IF;

	// AS Block 31 - TRI_TO_H2O2
	IF gCMD_LR[IdxSkids_LR].Write_TRI_TO_H2O2.Send THEN
		gCMD_LR[IdxSkids_LR].Write_TRI_TO_H2O2.wTRI_TO_H2O2_SWAPPED := IDEC_REAL_Conv(gCMD_LR[IdxSkids_LR].Write_TRI_TO_H2O2.wTRI_TO_H2O2);
		MasterConfig_LR[IdxSkids_LR].action_enable[30].single := TRUE;
		MasterConfig_LR[IdxSkids_LR].action_enable[71].single := TRUE; // Send Recalculation Command
		gCMD_LR[IdxSkids_LR].Write_TRI_TO_H2O2.Send := FALSE;
	END_IF;

	// AS Block 32 - PMAX_HOA
	IF gCMD_LR[IdxSkids_LR].Write_PMAX_HOA.Send THEN
		gCMD_LR[IdxSkids_LR].Write_PMAX_HOA.wPMAX_HOA := STRING_TO_UINT(gCMD_LR[IdxSkids_LR].Write_PMAX_HOA.wPMAX_HOA_String);
		MasterConfig_LR[IdxSkids_LR].action_enable[31].single := TRUE;
		gCMD_LR[IdxSkids_LR].Write_PMAX_HOA.Send := FALSE;
	ELSIF NOT gVis.Main.Out.DialogOpen THEN
		gCMD_LR[IdxSkids_LR].Write_PMAX_HOA.wPMAX_HOA_String := UINT_TO_STRING(gSkid_LR[IdxSkids_LR].Pmax_General_Variables.PMAX_HOA);
	END_IF;

	// AS Block 33 - PMAX_CONC
	IF gCMD_LR[IdxSkids_LR].Write_PMAX_CONC.Send THEN
		gCMD_LR[IdxSkids_LR].Write_PMAX_CONC.wPMAX_CONC_SWAPPED := IDEC_REAL_Conv(gCMD_LR[IdxSkids_LR].Write_PMAX_CONC.wPMAX_CONC);
		MasterConfig_LR[IdxSkids_LR].action_enable[32].single := TRUE;
		MasterConfig_LR[IdxSkids_LR].action_enable[71].single := TRUE; // Send Recalculation Command
		gCMD_LR[IdxSkids_LR].Write_PMAX_CONC.Send := FALSE;
	END_IF;

	// AS Block 34 - HP_CONC
	IF gCMD_LR[IdxSkids_LR].Write_HP_CONC.Send THEN
		gCMD_LR[IdxSkids_LR].Write_HP_CONC.wHP_CONC_SWAPPED := IDEC_REAL_Conv(gCMD_LR[IdxSkids_LR].Write_HP_CONC.wHP_CONC);
		MasterConfig_LR[IdxSkids_LR].action_enable[33].single := TRUE;
		MasterConfig_LR[IdxSkids_LR].action_enable[71].single := TRUE; // Send Recalculation Command
		gCMD_LR[IdxSkids_LR].Write_HP_CONC.Send := FALSE;
	END_IF;

	// AS Block 35 - NAOH_CONC
	IF gCMD_LR[IdxSkids_LR].Write_NAOH_CONC.Send THEN
		gCMD_LR[IdxSkids_LR].Write_NAOH_CONC.wNAOH_CONC_SWAPPED := IDEC_REAL_Conv(gCMD_LR[IdxSkids_LR].Write_NAOH_CONC.wNAOH_CONC);
		MasterConfig_LR[IdxSkids_LR].action_enable[34].single := TRUE;
		MasterConfig_LR[IdxSkids_LR].action_enable[71].single := TRUE; // Send Recalculation Command
		gCMD_LR[IdxSkids_LR].Write_NAOH_CONC.Send := FALSE;
	END_IF;

	// AS Block 36 - P101_STRT_CMD
	IF gCMD_LR[IdxSkids_LR].Write_P101_STRT_CMD.Send THEN
		MasterConfig_LR[IdxSkids_LR].action_enable[35].single := TRUE;
		gCMD_LR[IdxSkids_LR].Write_P101_STRT_CMD.Send := FALSE;
	END_IF;

	// AS Block 37 - P101_STP_CMD
	IF gCMD_LR[IdxSkids_LR].Write_P101_STP_CMD.Send THEN
		MasterConfig_LR[IdxSkids_LR].action_enable[36].single := TRUE;
		gCMD_LR[IdxSkids_LR].Write_P101_STP_CMD.Send := FALSE;
	END_IF;

	// AS Block 38 - P101_SP
	IF gCMD_LR[IdxSkids_LR].Write_P101_SP.Send THEN
		gCMD_LR[IdxSkids_LR].Write_P101_SP.wP101_SP_SWAPPED := IDEC_REAL_Conv(gCMD_LR[IdxSkids_LR].Write_P101_SP.wP101_SP);
		MasterConfig_LR[IdxSkids_LR].action_enable[37].single := TRUE;
		gCMD_LR[IdxSkids_LR].Write_P101_SP.Send := FALSE;
	END_IF;

	// AS Block 39 - P102_STRT_CMD
	IF gCMD_LR[IdxSkids_LR].Write_P102_STRT_CMD.Send THEN
		MasterConfig_LR[IdxSkids_LR].action_enable[38].single := TRUE;
		gCMD_LR[IdxSkids_LR].Write_P102_STRT_CMD.Send := FALSE;
	END_IF;

	// AS Block 40 - P102_STP_CMD
	IF gCMD_LR[IdxSkids_LR].Write_P102_STP_CMD.Send THEN
		MasterConfig_LR[IdxSkids_LR].action_enable[39].single := TRUE;
		gCMD_LR[IdxSkids_LR].Write_P102_STP_CMD.Send := FALSE;
	END_IF;

	// AS Block 41 - P102_SP
	IF gCMD_LR[IdxSkids_LR].Write_P102_SP.Send THEN
		gCMD_LR[IdxSkids_LR].Write_P102_SP.wP102_SP_SWAPPED := IDEC_REAL_Conv(gCMD_LR[IdxSkids_LR].Write_P102_SP.wP102_SP);
		MasterConfig_LR[IdxSkids_LR].action_enable[40].single := TRUE;
		gCMD_LR[IdxSkids_LR].Write_P102_SP.Send := FALSE;
	END_IF;

	// AS Block 42 - P103_STRT_CMD
	IF gCMD_LR[IdxSkids_LR].Write_P103_STRT_CMD.Send THEN
		MasterConfig_LR[IdxSkids_LR].action_enable[41].single := TRUE;
		gCMD_LR[IdxSkids_LR].Write_P103_STRT_CMD.Send := FALSE;
	END_IF;

	// AS Block 43 - P103_STP_CMD
	IF gCMD_LR[IdxSkids_LR].Write_P103_STP_CMD.Send THEN
		MasterConfig_LR[IdxSkids_LR].action_enable[42].single := TRUE;
		gCMD_LR[IdxSkids_LR].Write_P103_STP_CMD.Send := FALSE;
	END_IF;

	// AS Block 44 - P103_SP
	IF gCMD_LR[IdxSkids_LR].Write_P103_SP.Send THEN
		gCMD_LR[IdxSkids_LR].Write_P103_SP.wP103_SP_SWAPPED := IDEC_REAL_Conv(gCMD_LR[IdxSkids_LR].Write_P103_SP.wP103_SP);
		MasterConfig_LR[IdxSkids_LR].action_enable[43].single := TRUE;
		gCMD_LR[IdxSkids_LR].Write_P103_SP.Send := FALSE;
	END_IF;

	// AS Block 45 - P104_STRT_CMD
	IF gCMD_LR[IdxSkids_LR].Write_P104_STRT_CMD.Send THEN
		MasterConfig_LR[IdxSkids_LR].action_enable[44].single := TRUE;
		gCMD_LR[IdxSkids_LR].Write_P104_STRT_CMD.Send := FALSE;
	END_IF;

	// AS Block 46 - P104_STP_CMD
	IF gCMD_LR[IdxSkids_LR].Write_P104_STP_CMD.Send THEN
		MasterConfig_LR[IdxSkids_LR].action_enable[45].single := TRUE;
		gCMD_LR[IdxSkids_LR].Write_P104_STP_CMD.Send := FALSE;
	END_IF;

	// AS Block 47 - P104_SP
	IF gCMD_LR[IdxSkids_LR].Write_P104_SP.Send THEN
		gCMD_LR[IdxSkids_LR].Write_P104_SP.wP104_SP_SWAPPED := IDEC_REAL_Conv(gCMD_LR[IdxSkids_LR].Write_P104_SP.wP104_SP);
		MasterConfig_LR[IdxSkids_LR].action_enable[46].single := TRUE;
		gCMD_LR[IdxSkids_LR].Write_P104_SP.Send := FALSE;
	END_IF;

	// AS Block 48 is a READ block

	// AS Block 49 - LOCK_CMD
	IF gCMD_LR[IdxSkids_LR].Write_LOCK_CMD.Send THEN
		MasterConfig_LR[IdxSkids_LR].action_enable[48].single := TRUE;
		gCMD_LR[IdxSkids_LR].Write_LOCK_CMD.Send := FALSE;
	END_IF;

	// AS Block 50 - UNLOCK_CMD
	IF gCMD_LR[IdxSkids_LR].Write_UNLOCK_CMD.Send THEN
		MasterConfig_LR[IdxSkids_LR].action_enable[49].single := TRUE;
		gCMD_LR[IdxSkids_LR].Write_UNLOCK_CMD.Send := FALSE;
	END_IF;

	// AS Block 51 - FI301_SIM_CMD
	IF gCMD_LR[IdxSkids_LR].Write_FI301_SIM_CMD.Send THEN
		MasterConfig_LR[IdxSkids_LR].action_enable[50].single := TRUE;
		gCMD_LR[IdxSkids_LR].Write_FI301_SIM_CMD.Send := FALSE;
	END_IF;

	// AS Block 52 - FI301_MEA_CMD
	IF gCMD_LR[IdxSkids_LR].Write_FI301_MEA_CMD.Send THEN
		MasterConfig_LR[IdxSkids_LR].action_enable[51].single := TRUE;
		gCMD_LR[IdxSkids_LR].Write_FI301_MEA_CMD.Send := FALSE;
	END_IF;

	// AS Block 53 - FI301_SIM
	IF gCMD_LR[IdxSkids_LR].Write_FI301_SIM.Send THEN
		gCMD_LR[IdxSkids_LR].Write_FI301_SIM.wFI301_SIM_SWAPPED := IDEC_REAL_Conv(gCMD_LR[IdxSkids_LR].Write_FI301_SIM.wFI301_SIM);
		MasterConfig_LR[IdxSkids_LR].action_enable[52].single := TRUE;
		gCMD_LR[IdxSkids_LR].Write_FI301_SIM.Send := FALSE;
	END_IF;

	// AS Block 54 - FI302_SIM_CMD
	IF gCMD_LR[IdxSkids_LR].Write_FI302_SIM_CMD.Send THEN
		MasterConfig_LR[IdxSkids_LR].action_enable[53].single := TRUE;
		gCMD_LR[IdxSkids_LR].Write_FI302_SIM_CMD.Send := FALSE;
	END_IF;

	// AS Block 55 - FI302_MEA_CMD
	IF gCMD_LR[IdxSkids_LR].Write_FI302_MEA_CMD.Send THEN
		MasterConfig_LR[IdxSkids_LR].action_enable[54].single := TRUE;
		gCMD_LR[IdxSkids_LR].Write_FI302_MEA_CMD.Send := FALSE;
	END_IF;

	// AS Block 56 - FI302_SIM
	IF gCMD_LR[IdxSkids_LR].Write_FI302_SIM.Send THEN
		gCMD_LR[IdxSkids_LR].Write_FI302_SIM.wFI302_SIM_SWAPPED := IDEC_REAL_Conv(gCMD_LR[IdxSkids_LR].Write_FI302_SIM.wFI302_SIM);
		MasterConfig_LR[IdxSkids_LR].action_enable[55].single := TRUE;
		gCMD_LR[IdxSkids_LR].Write_FI302_SIM.Send := FALSE;
	END_IF;

	// AS Block 57 - FI303_SIM_CMD
	IF gCMD_LR[IdxSkids_LR].Write_FI303_SIM_CMD.Send THEN
		MasterConfig_LR[IdxSkids_LR].action_enable[56].single := TRUE;
		gCMD_LR[IdxSkids_LR].Write_FI303_SIM_CMD.Send := FALSE;
	END_IF;

	// AS Block 58 - FI303_MEA_CMD
	IF gCMD_LR[IdxSkids_LR].Write_FI303_MEA_CMD.Send THEN
		MasterConfig_LR[IdxSkids_LR].action_enable[57].single := TRUE;
		gCMD_LR[IdxSkids_LR].Write_FI303_MEA_CMD.Send := FALSE;
	END_IF;

	// AS Block 59 - FI303_SIM
	IF gCMD_LR[IdxSkids_LR].Write_FI303_SIM.Send THEN
		gCMD_LR[IdxSkids_LR].Write_FI303_SIM.wFI303_SIM_SWAPPED := IDEC_REAL_Conv(gCMD_LR[IdxSkids_LR].Write_FI303_SIM.wFI303_SIM);
		MasterConfig_LR[IdxSkids_LR].action_enable[58].single := TRUE;
		gCMD_LR[IdxSkids_LR].Write_FI303_SIM.Send := FALSE;
	END_IF;

	// AS Block 60 - UNIT_ACK - RESET OF CONDITION PERFORMED IN MAIN.ST ALARMS RESET
	IF gVis.Main.In.AckAllAlarms_Skid_LR[IdxSkids_LR] THEN
		MasterConfig_LR[IdxSkids_LR].action_enable[59].single := TRUE;
	END_IF;

	// AS Block 61 IS THE TEXT READ INT BLOCK

	// AS Block 62 - XV101_OPEN_CMD
	IF gCMD_LR[IdxSkids_LR].Write_XV101_OPEN_CMD.Send THEN
		MasterConfig_LR[IdxSkids_LR].action_enable[61].single := TRUE;
		gCMD_LR[IdxSkids_LR].Write_XV101_OPEN_CMD.Send := FALSE;
	END_IF;

	// AS Block 63 - XV102_OPEN_CMD
	IF gCMD_LR[IdxSkids_LR].Write_XV102_OPEN_CMD.Send THEN
		MasterConfig_LR[IdxSkids_LR].action_enable[62].single := TRUE;
		gCMD_LR[IdxSkids_LR].Write_XV102_OPEN_CMD.Send := FALSE;
	END_IF;

	// AS Block 64 - XV103_OPEN_CMD
	IF gCMD_LR[IdxSkids_LR].Write_XV103_OPEN_CMD.Send THEN
		MasterConfig_LR[IdxSkids_LR].action_enable[63].single := TRUE;
		gCMD_LR[IdxSkids_LR].Write_XV103_OPEN_CMD.Send := FALSE;
	END_IF;

	// AS Block 65 - XV104_OPEN_CMD
	IF gCMD_LR[IdxSkids_LR].Write_XV104_OPEN_CMD.Send THEN
		MasterConfig_LR[IdxSkids_LR].action_enable[64].single := TRUE;
		gCMD_LR[IdxSkids_LR].Write_XV104_OPEN_CMD.Send := FALSE;
	END_IF;

	// AS Block 66 - XV201_OPEN_CMD
	IF gCMD_LR[IdxSkids_LR].Write_XV201_OPEN_CMD.Send THEN
		MasterConfig_LR[IdxSkids_LR].action_enable[65].single := TRUE;
		gCMD_LR[IdxSkids_LR].Write_XV201_OPEN_CMD.Send := FALSE;
	END_IF;

	// AS Block 67 - XV202_OPEN_CMD
	IF gCMD_LR[IdxSkids_LR].Write_XV202_OPEN_CMD.Send THEN
		MasterConfig_LR[IdxSkids_LR].action_enable[66].single := TRUE;
		gCMD_LR[IdxSkids_LR].Write_XV202_OPEN_CMD.Send := FALSE;
	END_IF;

	// AS Block 68 - XV203_OPEN_CMD
	IF gCMD_LR[IdxSkids_LR].Write_XV203_OPEN_CMD.Send THEN
		MasterConfig_LR[IdxSkids_LR].action_enable[67].single := TRUE;
		gCMD_LR[IdxSkids_LR].Write_XV203_OPEN_CMD.Send := FALSE;
	END_IF;

	// AS Block 69 - AS_USER
	IF gCMD_LR[IdxSkids_LR].Write_AS_USER.Send THEN
		MasterConfig_LR[IdxSkids_LR].action_enable[68].single := TRUE;
		gCMD_LR[IdxSkids_LR].Write_AS_USER.Send := FALSE;
	END_IF;

	// AS Block 70 - AS_ACCESS
	IF gCMD_LR[IdxSkids_LR].Write_AS_ACCESS.Send THEN
		MasterConfig_LR[IdxSkids_LR].action_enable[69].single := TRUE;
		gCMD_LR[IdxSkids_LR].Write_AS_ACCESS.Send := FALSE;
	END_IF;

	// AS Block 71 - TOTALIZER_RESET
	IF gCMD_LR[IdxSkids_LR].Write_TOTALIZER_RESET.Send THEN
		MasterConfig_LR[IdxSkids_LR].action_enable[70].single := TRUE;
		gCMD_LR[IdxSkids_LR].Write_TOTALIZER_RESET.Send := FALSE;
	END_IF;

	// AS Block 72 - RECALC_CMD - Sends With Changes to Settings Above

	// AS Block 73 - ESTOP
	IF gCMD_LR[IdxSkids_LR].Write_ESTOP.Send THEN
		MasterConfig_LR[IdxSkids_LR].action_enable[72].single := TRUE;
		gCMD_LR[IdxSkids_LR].Write_ESTOP.Send := FALSE;
	END_IF;

	///////////////////////////////////////////

	// AS Block 74 - P101_AUTOCAL
	IF gCMD_LR[IdxSkids_LR].Write_P101_AUTOCAL.Send THEN
		MasterConfig_LR[IdxSkids_LR].action_enable[73].single := TRUE;
		gCMD_LR[IdxSkids_LR].Write_P101_AUTOCAL.Send := FALSE;
	END_IF;

	// AS Block 75 - P101_GAIN
	IF gCMD_LR[IdxSkids_LR].Write_P101_GAIN.Send THEN
		gCMD_LR[IdxSkids_LR].Write_P101_GAIN.wP101_GAIN_SWAPPED := IDEC_REAL_Conv(gCMD_LR[IdxSkids_LR].Write_P101_GAIN.wP101_GAIN);
		MasterConfig_LR[IdxSkids_LR].action_enable[74].single := TRUE;
		gCMD_LR[IdxSkids_LR].Write_P101_GAIN.Send := FALSE;
	END_IF;

	// AS Block 76 - P101_STEPADJ
	IF gCMD_LR[IdxSkids_LR].Write_P101_STEPADJ.Send THEN
		gCMD_LR[IdxSkids_LR].Write_P101_STEPADJ.wP101_STEPADJ_SWAPPED := IDEC_REAL_Conv(gCMD_LR[IdxSkids_LR].Write_P101_STEPADJ.wP101_STEPADJ);
		MasterConfig_LR[IdxSkids_LR].action_enable[75].single := TRUE;
		gCMD_LR[IdxSkids_LR].Write_P101_STEPADJ.Send := FALSE;
	END_IF;

	// AS Block 77 - P101_TOTALADJ
	IF gCMD_LR[IdxSkids_LR].Write_P101_TOTALADJ.Send THEN
		gCMD_LR[IdxSkids_LR].Write_P101_TOTALADJ.wP101_TOTALADJ_SWAPPED := IDEC_REAL_Conv(gCMD_LR[IdxSkids_LR].Write_P101_TOTALADJ.wP101_TOTALADJ);
		MasterConfig_LR[IdxSkids_LR].action_enable[76].single := TRUE;
		gCMD_LR[IdxSkids_LR].Write_P101_TOTALADJ.Send := FALSE;
	END_IF;

	// AS Block 78 - P102_AUTOCAL
	IF gCMD_LR[IdxSkids_LR].Write_P102_AUTOCAL.Send THEN
		MasterConfig_LR[IdxSkids_LR].action_enable[77].single := TRUE;
		gCMD_LR[IdxSkids_LR].Write_P102_AUTOCAL.Send := FALSE;
	END_IF;

	// AS Block 79 - P102_AUTOFLO_ADPT
	IF gCMD_LR[IdxSkids_LR].Write_P102_AUTOFLO_ADPT.Send THEN
		MasterConfig_LR[IdxSkids_LR].action_enable[78].single := TRUE;
		gCMD_LR[IdxSkids_LR].Write_P102_AUTOFLO_ADPT.Send := FALSE;
	END_IF;

	// AS Block 80 - P102_GAIN
	IF gCMD_LR[IdxSkids_LR].Write_P102_GAIN.Send THEN
		gCMD_LR[IdxSkids_LR].Write_P102_GAIN.wP102_GAIN_SWAPPED := IDEC_REAL_Conv(gCMD_LR[IdxSkids_LR].Write_P102_GAIN.wP102_GAIN);
		MasterConfig_LR[IdxSkids_LR].action_enable[79].single := TRUE;
		gCMD_LR[IdxSkids_LR].Write_P102_GAIN.Send := FALSE;
	END_IF;

	// AS Block 81 - P102_STEPADJ
	IF gCMD_LR[IdxSkids_LR].Write_P102_STEPADJ.Send THEN
		gCMD_LR[IdxSkids_LR].Write_P102_STEPADJ.wP102_STEPADJ_SWAPPED := IDEC_REAL_Conv(gCMD_LR[IdxSkids_LR].Write_P102_STEPADJ.wP102_STEPADJ);
		MasterConfig_LR[IdxSkids_LR].action_enable[80].single := TRUE;
		gCMD_LR[IdxSkids_LR].Write_P102_STEPADJ.Send := FALSE;
	END_IF;

	// AS Block 82 - P102_TOTALADJ
	IF gCMD_LR[IdxSkids_LR].Write_P102_TOTALADJ.Send THEN
		gCMD_LR[IdxSkids_LR].Write_P102_TOTALADJ.wP102_TOTALADJ_SWAPPED := IDEC_REAL_Conv(gCMD_LR[IdxSkids_LR].Write_P102_TOTALADJ.wP102_TOTALADJ);
		MasterConfig_LR[IdxSkids_LR].action_enable[81].single := TRUE;
		gCMD_LR[IdxSkids_LR].Write_P102_TOTALADJ.Send := FALSE;
	END_IF;

	// AS Block 83 - P103_AUTOCAL
	IF gCMD_LR[IdxSkids_LR].Write_P103_AUTOCAL.Send THEN
		MasterConfig_LR[IdxSkids_LR].action_enable[82].single := TRUE;
		gCMD_LR[IdxSkids_LR].Write_P103_AUTOCAL.Send := FALSE;
	END_IF;

	// AS Block 84 - P103_AUTOFLO_ADPT
	IF gCMD_LR[IdxSkids_LR].Write_P103_AUTOFLO_ADPT.Send THEN
		MasterConfig_LR[IdxSkids_LR].action_enable[83].single := TRUE;
		gCMD_LR[IdxSkids_LR].Write_P103_AUTOFLO_ADPT.Send := FALSE;
	END_IF;

	// AS Block 85 - P103_GAIN
	IF gCMD_LR[IdxSkids_LR].Write_P103_GAIN.Send THEN
		gCMD_LR[IdxSkids_LR].Write_P103_GAIN.wP103_GAIN_SWAPPED := IDEC_REAL_Conv(gCMD_LR[IdxSkids_LR].Write_P103_GAIN.wP103_GAIN);
		MasterConfig_LR[IdxSkids_LR].action_enable[84].single := TRUE;
		gCMD_LR[IdxSkids_LR].Write_P103_GAIN.Send := FALSE;
	END_IF;

	// AS Block 86 - P103_STEPADJ
	IF gCMD_LR[IdxSkids_LR].Write_P103_STEPADJ.Send THEN
		gCMD_LR[IdxSkids_LR].Write_P103_STEPADJ.wP103_STEPADJ_SWAPPED := IDEC_REAL_Conv(gCMD_LR[IdxSkids_LR].Write_P103_STEPADJ.wP103_STEPADJ);
		MasterConfig_LR[IdxSkids_LR].action_enable[85].single := TRUE;
		gCMD_LR[IdxSkids_LR].Write_P103_STEPADJ.Send := FALSE;
	END_IF;

	// AS Block 87 - P103_TOTALADJ
	IF gCMD_LR[IdxSkids_LR].Write_P103_TOTALADJ.Send THEN
		gCMD_LR[IdxSkids_LR].Write_P103_TOTALADJ.wP103_TOTALADJ_SWAPPED := IDEC_REAL_Conv(gCMD_LR[IdxSkids_LR].Write_P103_TOTALADJ.wP103_TOTALADJ);
		MasterConfig_LR[IdxSkids_LR].action_enable[86].single := TRUE;
		gCMD_LR[IdxSkids_LR].Write_P103_TOTALADJ.Send := FALSE;
	END_IF;

	// AS Block 88 - P104_AUTOCAL
	IF gCMD_LR[IdxSkids_LR].Write_P104_AUTOCAL.Send THEN
		MasterConfig_LR[IdxSkids_LR].action_enable[87].single := TRUE;
		gCMD_LR[IdxSkids_LR].Write_P104_AUTOCAL.Send := FALSE;
	END_IF;

	// AS Block 89 - P104_AUTOCAL_PV
	IF gCMD_LR[IdxSkids_LR].Write_P104_AUTOCAL_PV.Send THEN
		MasterConfig_LR[IdxSkids_LR].action_enable[88].single := TRUE;
		gCMD_LR[IdxSkids_LR].Write_P104_AUTOCAL_PV.Send := FALSE;
	END_IF;

	// AS Block 90 - P104_AUTOFLO_ADPT
	IF gCMD_LR[IdxSkids_LR].Write_P104_AUTOFLO_ADPT.Send THEN
		MasterConfig_LR[IdxSkids_LR].action_enable[89].single := TRUE;
		gCMD_LR[IdxSkids_LR].Write_P104_AUTOFLO_ADPT.Send := FALSE;
	END_IF;

	// AS Block 91 - P104_GAIN
	IF gCMD_LR[IdxSkids_LR].Write_P104_GAIN.Send THEN
		gCMD_LR[IdxSkids_LR].Write_P104_GAIN.wP104_GAIN_SWAPPED := IDEC_REAL_Conv(gCMD_LR[IdxSkids_LR].Write_P104_GAIN.wP104_GAIN);
		MasterConfig_LR[IdxSkids_LR].action_enable[90].single := TRUE;
		gCMD_LR[IdxSkids_LR].Write_P104_GAIN.Send := FALSE;
	END_IF;

	// AS Block 92 - P104_STEPADJ
	IF gCMD_LR[IdxSkids_LR].Write_P104_STEPADJ.Send THEN
		gCMD_LR[IdxSkids_LR].Write_P104_STEPADJ.wP104_STEPADJ_SWAPPED := IDEC_REAL_Conv(gCMD_LR[IdxSkids_LR].Write_P104_STEPADJ.wP104_STEPADJ);
		MasterConfig_LR[IdxSkids_LR].action_enable[91].single := TRUE;
		gCMD_LR[IdxSkids_LR].Write_P104_STEPADJ.Send := FALSE;
	END_IF;

	// AS Block 93 - P104_TOTALADJ
	IF gCMD_LR[IdxSkids_LR].Write_P104_TOTALADJ.Send THEN
		gCMD_LR[IdxSkids_LR].Write_P104_TOTALADJ.wP104_TOTALADJ_SWAPPED := IDEC_REAL_Conv(gCMD_LR[IdxSkids_LR].Write_P104_TOTALADJ.wP104_TOTALADJ);
		MasterConfig_LR[IdxSkids_LR].action_enable[92].single := TRUE;
		gCMD_LR[IdxSkids_LR].Write_P104_TOTALADJ.Send := FALSE;
	END_IF;

	// AS Block 94 - P201_AUTOCAL
	IF gCMD_LR[IdxSkids_LR].Write_P201_AUTOCAL.Send THEN
		MasterConfig_LR[IdxSkids_LR].action_enable[93].single := TRUE;
		gCMD_LR[IdxSkids_LR].Write_P201_AUTOCAL.Send := FALSE;
	END_IF;

	// AS Block 95 - P201_AUTOCAL_PV
	IF gCMD_LR[IdxSkids_LR].Write_P201_AUTOCAL_PV.Send THEN
		MasterConfig_LR[IdxSkids_LR].action_enable[94].single := TRUE;
		gCMD_LR[IdxSkids_LR].Write_P201_AUTOCAL_PV.Send := FALSE;
	END_IF;

	// AS Block 96 - P201_AUTOFLO_ADPT
	IF gCMD_LR[IdxSkids_LR].Write_P201_AUTOFLO_ADPT.Send THEN
		MasterConfig_LR[IdxSkids_LR].action_enable[95].single := TRUE;
		gCMD_LR[IdxSkids_LR].Write_P201_AUTOFLO_ADPT.Send := FALSE;
	END_IF;

	// AS Block 97 - P201_GAIN
	IF gCMD_LR[IdxSkids_LR].Write_P201_GAIN.Send THEN
		gCMD_LR[IdxSkids_LR].Write_P201_GAIN.wP201_GAIN_SWAPPED := IDEC_REAL_Conv(gCMD_LR[IdxSkids_LR].Write_P201_GAIN.wP201_GAIN);
		MasterConfig_LR[IdxSkids_LR].action_enable[96].single := TRUE;
		gCMD_LR[IdxSkids_LR].Write_P201_GAIN.Send := FALSE;
	END_IF;

	// AS Block 98 - P201_STEPADJ
	IF gCMD_LR[IdxSkids_LR].Write_P201_STEPADJ.Send THEN
		gCMD_LR[IdxSkids_LR].Write_P201_STEPADJ.wP201_STEPADJ_SWAPPED := IDEC_REAL_Conv(gCMD_LR[IdxSkids_LR].Write_P201_STEPADJ.wP201_STEPADJ);
		MasterConfig_LR[IdxSkids_LR].action_enable[97].single := TRUE;
		gCMD_LR[IdxSkids_LR].Write_P201_STEPADJ.Send := FALSE;
	END_IF;

	// AS Block 99 - P201_TOTALADJ
	IF gCMD_LR[IdxSkids_LR].Write_P201_TOTALADJ.Send THEN
		gCMD_LR[IdxSkids_LR].Write_P201_TOTALADJ.wP201_TOTALADJ_SWAPPED := IDEC_REAL_Conv(gCMD_LR[IdxSkids_LR].Write_P201_TOTALADJ.wP201_TOTALADJ);
		MasterConfig_LR[IdxSkids_LR].action_enable[98].single := TRUE;
		gCMD_LR[IdxSkids_LR].Write_P201_TOTALADJ.Send := FALSE;
	END_IF;

	// AS Block 100 - P202_AUTOCAL
	IF gCMD_LR[IdxSkids_LR].Write_P202_AUTOCAL.Send THEN
		MasterConfig_LR[IdxSkids_LR].action_enable[99].single := TRUE;
		gCMD_LR[IdxSkids_LR].Write_P202_AUTOCAL.Send := FALSE;
	END_IF;

	// AS Block 101 - P202_AUTOCAL_PV
	IF gCMD_LR[IdxSkids_LR].Write_P202_AUTOCAL_PV.Send THEN
		MasterConfig_LR[IdxSkids_LR].action_enable[100].single := TRUE;
		gCMD_LR[IdxSkids_LR].Write_P202_AUTOCAL_PV.Send := FALSE;
	END_IF;

	// AS Block 102 - P202_AUTOFLO_ADPT
	IF gCMD_LR[IdxSkids_LR].Write_P202_AUTOFLO_ADPT.Send THEN
		MasterConfig_LR[IdxSkids_LR].action_enable[101].single := TRUE;
		gCMD_LR[IdxSkids_LR].Write_P202_AUTOFLO_ADPT.Send := FALSE;
	END_IF;

	// AS Block 103 - P202_GAIN
	IF gCMD_LR[IdxSkids_LR].Write_P202_GAIN.Send THEN
		gCMD_LR[IdxSkids_LR].Write_P202_GAIN.wP202_GAIN_SWAPPED := IDEC_REAL_Conv(gCMD_LR[IdxSkids_LR].Write_P202_GAIN.wP202_GAIN);
		MasterConfig_LR[IdxSkids_LR].action_enable[102].single := TRUE;
		gCMD_LR[IdxSkids_LR].Write_P202_GAIN.Send := FALSE;
	END_IF;

	// AS Block 104 - P202_STEPADJ
	IF gCMD_LR[IdxSkids_LR].Write_P202_STEPADJ.Send THEN
		gCMD_LR[IdxSkids_LR].Write_P202_STEPADJ.wP202_STEPADJ_SWAPPED := IDEC_REAL_Conv(gCMD_LR[IdxSkids_LR].Write_P202_STEPADJ.wP202_STEPADJ);
		MasterConfig_LR[IdxSkids_LR].action_enable[103].single := TRUE;
		gCMD_LR[IdxSkids_LR].Write_P202_STEPADJ.Send := FALSE;
	END_IF;

	// AS Block 105 - P202_TOTALADJ
	IF gCMD_LR[IdxSkids_LR].Write_P202_TOTALADJ.Send THEN
		gCMD_LR[IdxSkids_LR].Write_P202_TOTALADJ.wP202_TOTALADJ_SWAPPED := IDEC_REAL_Conv(gCMD_LR[IdxSkids_LR].Write_P202_TOTALADJ.wP202_TOTALADJ);
		MasterConfig_LR[IdxSkids_LR].action_enable[104].single := TRUE;
		gCMD_LR[IdxSkids_LR].Write_P202_TOTALADJ.Send := FALSE;
	END_IF;

	// AS Block 106 - P203_AUTOCAL
	IF gCMD_LR[IdxSkids_LR].Write_P203_AUTOCAL.Send THEN
		MasterConfig_LR[IdxSkids_LR].action_enable[105].single := TRUE;
		gCMD_LR[IdxSkids_LR].Write_P203_AUTOCAL.Send := FALSE;
	END_IF;

	// AS Block 107 - P203_AUTOCAL_PV
	IF gCMD_LR[IdxSkids_LR].Write_P203_AUTOCAL_PV.Send THEN
		MasterConfig_LR[IdxSkids_LR].action_enable[106].single := TRUE;
		gCMD_LR[IdxSkids_LR].Write_P203_AUTOCAL_PV.Send := FALSE;
	END_IF;

	// AS Block 108 - P203_AUTOFLO_ADPT
	IF gCMD_LR[IdxSkids_LR].Write_P203_AUTOFLO_ADPT.Send THEN
		MasterConfig_LR[IdxSkids_LR].action_enable[107].single := TRUE;
		gCMD_LR[IdxSkids_LR].Write_P203_AUTOFLO_ADPT.Send := FALSE;
	END_IF;

	// AS Block 109 - P203_GAIN
	IF gCMD_LR[IdxSkids_LR].Write_P203_GAIN.Send THEN
		gCMD_LR[IdxSkids_LR].Write_P203_GAIN.wP203_GAIN_SWAPPED := IDEC_REAL_Conv(gCMD_LR[IdxSkids_LR].Write_P203_GAIN.wP203_GAIN);
		MasterConfig_LR[IdxSkids_LR].action_enable[108].single := TRUE;
		gCMD_LR[IdxSkids_LR].Write_P203_GAIN.Send := FALSE;
	END_IF;

	// AS Block 110 - P203_STEPADJ
	IF gCMD_LR[IdxSkids_LR].Write_P203_STEPADJ.Send THEN
		gCMD_LR[IdxSkids_LR].Write_P203_STEPADJ.wP203_STEPADJ_SWAPPED := IDEC_REAL_Conv(gCMD_LR[IdxSkids_LR].Write_P203_STEPADJ.wP203_STEPADJ);
		MasterConfig_LR[IdxSkids_LR].action_enable[109].single := TRUE;
		gCMD_LR[IdxSkids_LR].Write_P203_STEPADJ.Send := FALSE;
	END_IF;

	// AS Block 111 - P203_TOTALADJ
	IF gCMD_LR[IdxSkids_LR].Write_P203_TOTALADJ.Send THEN
		gCMD_LR[IdxSkids_LR].Write_P203_TOTALADJ.wP203_TOTALADJ_SWAPPED := IDEC_REAL_Conv(gCMD_LR[IdxSkids_LR].Write_P203_TOTALADJ.wP203_TOTALADJ);
		MasterConfig_LR[IdxSkids_LR].action_enable[110].single := TRUE;
		gCMD_LR[IdxSkids_LR].Write_P203_TOTALADJ.Send := FALSE;
	END_IF;

	// AS Block 112 - USER ADMIN RESET
	IF gCMD_LR[IdxSkids_LR].Write_USERADMIN_RESET.Send THEN
		MasterConfig_LR[IdxSkids_LR].action_enable[111].single := TRUE;
		gCMD_LR[IdxSkids_LR].Write_USERADMIN_RESET.Send := FALSE;
	END_IF;

	// AS Block 113 - ROSTER1_PHONE
	IF gCMD_LR[IdxSkids_LR].Write_PHONE_INPUT1.Send THEN
		MasterConfig_LR[IdxSkids_LR].action_enable[112].single := TRUE;
		gCMD_LR[IdxSkids_LR].Write_PHONE_INPUT1.Send := FALSE;
	END_IF;

	// AS Block 114 - ROSTER2_PHONE
	IF gCMD_LR[IdxSkids_LR].Write_PHONE_INPUT2.Send THEN
		MasterConfig_LR[IdxSkids_LR].action_enable[113].single := TRUE;
		gCMD_LR[IdxSkids_LR].Write_PHONE_INPUT2.Send := FALSE;
	END_IF;

	// AS Block 115 - ROSTER3_PHONE
	IF gCMD_LR[IdxSkids_LR].Write_PHONE_INPUT3.Send THEN
		MasterConfig_LR[IdxSkids_LR].action_enable[114].single := TRUE;
		gCMD_LR[IdxSkids_LR].Write_PHONE_INPUT3.Send := FALSE;
	END_IF;

	// AS Block 116 - ROSTER4_PHONE
	IF gCMD_LR[IdxSkids_LR].Write_PHONE_INPUT4.Send THEN
		MasterConfig_LR[IdxSkids_LR].action_enable[115].single := TRUE;
		gCMD_LR[IdxSkids_LR].Write_PHONE_INPUT4.Send := FALSE;
	END_IF;

	// AS Block 117 - ROSTER5_PHONE
	IF gCMD_LR[IdxSkids_LR].Write_PHONE_INPUT5.Send THEN
		MasterConfig_LR[IdxSkids_LR].action_enable[116].single := TRUE;
		gCMD_LR[IdxSkids_LR].Write_PHONE_INPUT5.Send := FALSE;
	END_IF;

	// AS Block 118 - ROSTER6_PHONE
	IF gCMD_LR[IdxSkids_LR].Write_PHONE_INPUT6.Send THEN
		MasterConfig_LR[IdxSkids_LR].action_enable[117].single := TRUE;
		gCMD_LR[IdxSkids_LR].Write_PHONE_INPUT6.Send := FALSE;
	END_IF;

	// AS Block 119 - ROSTER7_PHONE
	IF gCMD_LR[IdxSkids_LR].Write_PHONE_INPUT7.Send THEN
		MasterConfig_LR[IdxSkids_LR].action_enable[118].single := TRUE;
		gCMD_LR[IdxSkids_LR].Write_PHONE_INPUT7.Send := FALSE;
	END_IF;

	// AS Block 120 - ROSTER8_PHONE
	IF gCMD_LR[IdxSkids_LR].Write_PHONE_INPUT8.Send THEN
		MasterConfig_LR[IdxSkids_LR].action_enable[119].single := TRUE;
		gCMD_LR[IdxSkids_LR].Write_PHONE_INPUT8.Send := FALSE;
	END_IF;

	// AS BLOCK 121 - ROSTER1_ENABLE
	IF gCMD_LR[IdxSkids_LR].Write_ENABLE_ROSTER1.Send THEN
		MasterConfig_LR[IdxSkids_LR].action_enable[120].single := TRUE;
		gCMD_LR[IdxSkids_LR].Write_ENABLE_ROSTER1.Send := FALSE;
	END_IF;

	// AS BLOCK 122 - ROSTER2_ENABLE
	IF gCMD_LR[IdxSkids_LR].Write_ENABLE_ROSTER2.Send THEN
		MasterConfig_LR[IdxSkids_LR].action_enable[121].single := TRUE;
		gCMD_LR[IdxSkids_LR].Write_ENABLE_ROSTER2.Send := FALSE;
	END_IF;

	// AS BLOCK 123 - ROSTER3_ENABLE
	IF gCMD_LR[IdxSkids_LR].Write_ENABLE_ROSTER3.Send THEN
		MasterConfig_LR[IdxSkids_LR].action_enable[122].single := TRUE;
		gCMD_LR[IdxSkids_LR].Write_ENABLE_ROSTER3.Send := FALSE;
	END_IF;

	// AS BLOCK 124 - ROSTER4_ENABLE
	IF gCMD_LR[IdxSkids_LR].Write_ENABLE_ROSTER4.Send THEN
		MasterConfig_LR[IdxSkids_LR].action_enable[123].single := TRUE;
		gCMD_LR[IdxSkids_LR].Write_ENABLE_ROSTER4.Send := FALSE;
	END_IF;

	// AS BLOCK 125 - ROSTER5_ENABLE
	IF gCMD_LR[IdxSkids_LR].Write_ENABLE_ROSTER5.Send THEN
		MasterConfig_LR[IdxSkids_LR].action_enable[124].single := TRUE;
		gCMD_LR[IdxSkids_LR].Write_ENABLE_ROSTER5.Send := FALSE;
	END_IF;

	// AS BLOCK 126 - ROSTER6_ENABLE
	IF gCMD_LR[IdxSkids_LR].Write_ENABLE_ROSTER6.Send THEN
		MasterConfig_LR[IdxSkids_LR].action_enable[125].single := TRUE;
		gCMD_LR[IdxSkids_LR].Write_ENABLE_ROSTER6.Send := FALSE;
	END_IF;

	// AS BLOCK 127 - ROSTER7_ENABLE
	IF gCMD_LR[IdxSkids_LR].Write_ENABLE_ROSTER7.Send THEN
		MasterConfig_LR[IdxSkids_LR].action_enable[126].single := TRUE;
		gCMD_LR[IdxSkids_LR].Write_ENABLE_ROSTER7.Send := FALSE;
	END_IF;

	// AS BLOCK 128 - ROSTER8_ENABLE
	IF gCMD_LR[IdxSkids_LR].Write_ENABLE_ROSTER8.Send THEN
		MasterConfig_LR[IdxSkids_LR].action_enable[127].single := TRUE;
		gCMD_LR[IdxSkids_LR].Write_ENABLE_ROSTER8.Send := FALSE;
	END_IF;

	// AS BLOCK 129 - AC_ALARM_ENABLE
	IF gCMD_LR[IdxSkids_LR].Write_AC_ALARM_ENABLE.Send THEN
		MasterConfig_LR[IdxSkids_LR].action_enable[128].single := TRUE;
		gCMD_LR[IdxSkids_LR].Write_AC_ALARM_ENABLE.Send := FALSE;
	END_IF;

	// AS BLOCK 130 - AC_TXT_ENABLE
	IF gCMD_LR[IdxSkids_LR].Write_AC_TXT_ENABLE.Send THEN
		MasterConfig_LR[IdxSkids_LR].action_enable[129].single := TRUE;
		gCMD_LR[IdxSkids_LR].Write_AC_TXT_ENABLE.Send := FALSE;
	END_IF;

	// AS BLOCK 131 - AC_ACTION
	IF gCMD_LR[IdxSkids_LR].Write_AC_ACTION.Send THEN
		MasterConfig_LR[IdxSkids_LR].action_enable[130].single := TRUE;
		gCMD_LR[IdxSkids_LR].Write_AC_ACTION.Send := FALSE;
	END_IF;

	// AS BLOCK 132 - AC_DELAY
	IF gCMD_LR[IdxSkids_LR].Write_AC_DELAY.Send THEN
		MasterConfig_LR[IdxSkids_LR].action_enable[131].single := TRUE;
		gCMD_LR[IdxSkids_LR].Write_AC_DELAY.Send := FALSE;
	END_IF;

	// AS BLOCK 133 - AC_OFFSET
	IF gCMD_LR[IdxSkids_LR].Write_AC_OFFSET.Send THEN
		MasterConfig_LR[IdxSkids_LR].action_enable[132].single := TRUE;
		gCMD_LR[IdxSkids_LR].Write_AC_OFFSET.Send := FALSE;
	END_IF;

	// AS Block 134 - AC_THRESHOLD
	IF gCMD_LR[IdxSkids_LR].Write_AC_THRESHOLD.Send THEN
		gCMD_LR[IdxSkids_LR].Write_AC_THRESHOLD.wAC_THRESHOLD_SWAPPED := IDEC_REAL_Conv(gCMD_LR[IdxSkids_LR].Write_AC_THRESHOLD.wAC_THRESHOLD);
		MasterConfig_LR[IdxSkids_LR].action_enable[133].single := TRUE;
		gCMD_LR[IdxSkids_LR].Write_AC_THRESHOLD.Send := FALSE;
	END_IF;

END_ACTION
```
